// TwinCAT 3 PLC project DemoPLC
// ProgramVersion: 3.1.4020.1
// libraries:
//   Tc2_Drive, * (Beckhoff Automation GmbH)
//   Tc2_EtherCAT, * (Beckhoff Automation GmbH)
//   Tc2_Math, * (Beckhoff Automation GmbH)
//   Tc2_MC2, * (Beckhoff Automation GmbH)
//   Tc2_MC2_Drive, * (Beckhoff Automation GmbH)
//   Tc2_MDP, * (Beckhoff Automation GmbH)
//   Tc2_Smtp, * (Beckhoff Automation GmbH)
//   Tc2_Standard, * (Beckhoff Automation GmbH)
//   Tc2_System, * (Beckhoff Automation GmbH)
//   Tc2_Utilities, * (Beckhoff Automation GmbH)
//   Tc3_Module, * (Beckhoff Automation GmbH)
// project tree:
//   DUTs/DataAndTime/ E_DayPL.TcDUT, E_DayPLShort.TcDUT, E_Location.TcDUT, E_MonthPL.TcDUT, E_SeasonPL.TcDUT, ST_Calendar.TcDUT, ST_ConstHoliday.TcDUT, ST_ConstLocation.TcDUT, ST_Holiday.TcDUT, ST_Location.TcDUT
//   DUTs/ GEN_MODE.TcDUT, NEWTYPE.TcDUT, ST_AX5000_Diag_MC2.TcDUT, ST_EL3403_Data.TcDUT, ST_KL3403_Report.TcDUT, ST_STRING_2040.TcDUT
//   / MAIN.TcPOU, PlcTask.TcTTO
//   POUs/Blinkers/ FB_Blink_AS.TcPOU, FB_Blink_S.TcPOU
//   POUs/Conversions/ ArrayOfReal_To_String.TcPOU, arrBOOL16_TO_WORD.TcPOU, arrBOOL8_TO_BYTE.TcPOU, ArrOfInt_To_String.TcPOU, FB_CONCAT_S2040.TcPOU, FB_IntTo2Byte.TcPOU, F_4BYTES_TO_DWORD.TcPOU, F_4BYTES_TO_REAL.TcPOU, F_8BYTES_TO_LREAL.TcPOU, F_BCDToDec.TcPOU, F_CLEAN_S2040.TcPOU, F_Convert_4BBCD_To_Real.TcPOU, F_DWORD_TO_REAL.TcPOU, F_Words_to_Real.TcPOU, GRAYB_TO_WORD.TcPOU, GRAYW_TO_WORD.TcPOU
//   POUs/Conversions/BitOriented/ BCD_TO_INT.TcPOU, F_1stByteW.TcPOU, F_1stByteWtoB.TcPOU, F_2Bytes_To_Word.TcPOU, F_2ndByteW.TcPOU, F_2ndByteWtoB.TcPOU, F_MaskWord.TcPOU, L_TBConvArrBitsToDword.TcPOU, L_TBConvBitsToByte.TcPOU, L_TBConvBitsToDword.TcPOU, L_TBConvBitsToWord.TcPOU, L_TBConvByteToBits.TcPOU, L_TBConvDwordToArrBits.TcPOU, L_TBConvDwordToBits.TcPOU, L_TBConvWordToBits.TcPOU, L_TBGetBitOfByte.TcPOU, L_TBGetBitOfDword.TcPOU, L_TBGetBitOfWord.TcPOU, L_TBResetBitOfByte.TcPOU, L_TBResetBitOfDword.TcPOU, L_TBResetBitOfWord.TcPOU, L_TBSetBitOfByte.TcPOU, L_TBSetBitOfDword.TcPOU, L_TBSetBitOfWord.TcPOU, L_TBSquareWave.TcPOU
//   POUs/DateAndTime/ FB_AstrTimeCET.TcPOU, FB_CycleTime.TcPOU, FB_DST.TcPOU, FB_GetSystemTime.TcPOU, FB_Period.TcPOU, FB_PolishPublicHoliday.TcPOU, FB_SimpleWorkTime.TcPOU, FB_TimeMeasure.TcPOU, FB_TimeMeasureEx.TcPOU, FB_WeekSchedule.TcPOU, FB_Worktime.TcPOU, FB_WorktimeCompact.TcPOU, F_DT_To_sDT_Ind.TcPOU, F_ExcelDateMin.TcPOU, F_ExcelDateSec.TcPOU, F_sDT_Ind_To_DT.TcPOU
//   POUs/EL_Terminals/ FB_EL3403.TcPOU, FB_EL3403Ex.TcPOU, FB_EL3403Ex2.TcPOU
//   POUs/FileAccess/ FB_EmailLog.TcPOU, FB_FileLog.TcPOU, FB_FilePutText.TcPOU, FB_ReceipRW.TcPOU, FB_SaveLineToFile.TcPOU, FB_SaveTextToFile.TcPOU (not stored), FB_WriteReportToFile.TcPOU, FB_XCopyCE.TcPOU
//   POUs/FlipFlop/ FB_toggle.TcPOU, FB_TOGGLE_WITH_RESET.TcPOU, FB_TypeJK.TcPOU, FB_TypeJK_SEL.TcPOU, FB_TypeRS.TcPOU, FB_TypeSR.TcPOU
//   POUs/HVAC/ FB_AirMixer.TcPOU, FB_Alarm.TcPOU, FB_Boiler_Load.TcPOU, FB_Controller2Point.TcPOU, FB_DeadNullRange.TcPOU, FB_LimitHVAC.TcPOU, FB_SeqCMH.TcPOU
//   POUs/KL_Terminals/ FB_KL320x_1channel.TcPOU, FB_KL32x8_1channel.TcPOU, FB_KL32x8_1channelEx.TcPOU, FB_KL3403_1channel.TcPOU, FB_PowerMeasuring.TcPOU
//   POUs/NC/ FB_AX5000_Diag_MC2.TcPOU, FB_AxisParameter.TcPOU, FB_CalculateSpeed.TcPOU, FB_Enc20bitToDWORD.TcPOU, FB_EncIntToDint.TcPOU, FB_EncWordtoDword.TcPOU, FB_ForceLockUnlock.TcPOU, FB_I2T_AX2000.TcPOU, FB_I2T_EL72x1.TcPOU, FB_PWM_BASIC.TcPOU, FB_SetBiasValue.TcPOU, FB_TorqueMonitoringEL_Ex2.TcPOU, FB_TorqueMonitoringEx2.TcPOU
//   POUs/Switches/ FB_2SwB.TcPOU, FB_2SwM.TcPOU, FB_Click.TcPOU, FB_ClickCounterBit.TcPOU, FB_ClickCounterByte.TcPOU, FB_Dimmer1P.TcPOU, FB_Dimmer1PMinMax.TcPOU, FB_Dimmer2P.TcPOU, FB_Dimmer2PMinMax.TcPOU, FB_ShortLong.TcPOU, FB_ShortLongTrig.TcPOU, FB_Sw4F.TcPOU, FB_Sw4FTrig.TcPOU, FB_SwOrSen.TcPOU, FB_SwOrSenTrig.TcPOU
//   POUs/Various/ FB_AnalogTo3Point.TcPOU, FB_Average.TcPOU, FB_CERHOST.TcPOU, FB_DiskFreeSpace.TcPOU, FB_Filter.TcPOU, FB_FilterEx.TcPOU, FB_Generator.TcPOU, FB_Hysteresis.TcPOU, FB_Persistent.TcPOU, FB_PIDBasic.TcPOU, FB_Ramp.TcPOU, FB_ReadRegister.TcPOU, FB_RecMove.TcPOU, FB_SetIPAddress.TcPOU, FB_SinGenerator.TcPOU, FB_WriteRegister.TcPOU, F_CRC_CALC.TcPOU, F_ScaleLREAL.TcPOU, F_Scaling.TcPOU (not stored), TIMER.TcPOU, TONR.TcPOU
// real-time tasks:
//   TASK PlcTask: cycle T#10ms, priority 20, ADS port 350

CONFIGURATION DemoPLC
    RESOURCE PLC ON TwinCAT3
        TASK PlcTask(INTERVAL := T#10ms, PRIORITY := 20);
        PROGRAM MAIN WITH PlcTask : MAIN;
    END_RESOURCE
END_CONFIGURATION

// ---- DUTs/DataAndTime/E_DayPL.TcDUT
TYPE E_DayPL :(Poniedzialek:=1, Wtorek, Sroda, Czwartek, Piatek, Sobota, Niedziela );
END_TYPE

// ---- DUTs/DataAndTime/E_DayPLShort.TcDUT
TYPE E_DayPLShort :(Pn:=1, Wt, SR, Cz, Pt, So, N);
END_TYPE

// ---- DUTs/DataAndTime/E_Location.TcDUT
TYPE E_Location : (Wroclaw:=1, Warszawa, Krakow, Zakopane, Katowice, Poznan );
END_TYPE

// ---- DUTs/DataAndTime/E_MonthPL.TcDUT
TYPE E_MonthPL :(Stycznen:=1, Luty, Marzec, Kwiecien, Maj,  Czerwiec, Lipiec, Sierpien, Wrzesien, Pazdziernik, Listopad, Grudzien);
END_TYPE

// ---- DUTs/DataAndTime/E_SeasonPL.TcDUT
TYPE E_SeasonPL : (Wiosna:=1, Lato, Jesien, Zima);
END_TYPE

// ---- DUTs/DataAndTime/ST_Calendar.TcDUT
TYPE ST_Calendar :
STRUCT
	dateDate : DATE;				(* data *)
	wYear : WORD;				(* rok  *)
	wMonth : WORD;				(* miesiąc  *)
	wDay : WORD;				(* dzień *)
	bLeapYear: BOOL;			(* true if rok przestępny *)
	eWeekDay: E_DayPL;			(* dzień tygodnia *)
	wNoWeek : WORD;			(* nr tygodnia w roku *)
	wDayInYear: WORD;			(* nr dnia w roku *)
	bHoliday : BOOL;				(* true jesli jest swieto *)
	sHolidayName: STRING(30);	(* nazwa swieta *)
	eSeason: E_SeasonPL;		(* pora roku *)
	sLocation: STRING(30);		(* lokalizacja *)
	rLatitude: REAL;				(* szerokosc geograficzna np. Wrocław :=51.1174 *) (* do obliczen wschodu i zachodu slonca *)
	rLongitude: REAL;				(* długosc geograficzna np. Wrocław := 17.0383 *)
	todSunRise: TOD;				(* sun_rise for current location *)
	todSunSet : TOD;				(* sun_set for current location *)
END_STRUCT
END_TYPE

// ---- DUTs/DataAndTime/ST_ConstHoliday.TcDUT
TYPE ST_ConstHoliday :
STRUCT
	// Zapamietane dni swiat 
	//  gc_ConstHoliday - rozmiar tablicy array of ST_Holiday size   -> Var_Global_Calendar;   
	//  w tablicy najpierw nalezy podac swieta stale 
	//  if month = 0 obliczamy swieto ruchome
	//  iExecute mowi ile dni wczesniej/pozniej jest swieto
	astLocation: ARRAY [1..15] OF ST_Holiday := [		(sName := 'Nowy Rok', 				wDay := 1, 	wMonth := 1),
														(sName := 'Swieto Pracy', 			wDay := 1, 	wMonth := 5),
														(sName := 'Konstytucja 3 Maja', 	wDay := 3, 	wMonth := 5),
														(sName := 'Wniebowstapienie NMP',	wDay := 15,	wMonth := 8),
														(sName := 'Wszystkich Swietych', 	wDay := 1, 	wMonth := 11),
														(sName := 'Swieto Niepodleglosc', 	wDay := 11, 	wMonth := 11),
														(sName := 'Boze Narodzenie', 		wDay := 25, 	wMonth := 12),
														(sName := 'Boze Narodzenie', 		wDay := 26, 	wMonth := 12),
														(sName := 'Wielki Piatek',			wDay := 0, 	wMonth := 0, iExecute := -2),
														(sName := 'Wielka Sobota', 			wDay := 0, 	wMonth := 0, iExecute := -1),
														(sName := 'Wielkanoc', 				wDay := 0, 	wMonth := 0, iExecute := 0),
														(sName := 'Poniedziałek Wielkanocny', wDay :=1,	wMonth := 0, iExecute := 1),
														(sName := 'Boze Cialo', 			wDay := 0, 	wMonth := 0, iExecute := 60),
														2(())];
END_STRUCT
END_TYPE

// ---- DUTs/DataAndTime/ST_ConstLocation.TcDUT
TYPE ST_ConstLocation :
STRUCT
	(* to memorize location *)
	(* gc_ConstLocation - max array of ST_Location  size  -> Var_Global_Calendar;   *)
	astLocation : ARRAY [1.. 10] OF ST_Location := [(sName := 'Wroclaw', rLatitude := 51.1174, rLongitude := 17.0383),
											(sName := 'Warszawa', rLatitude := 52.248, rLongitude := 21.008),
											(sName := 'Krakow', rLatitude := 50.085, rLongitude := 19.940),
											(sName := 'Zakopane', rLatitude := 49.3091, rLongitude := 19.9524),
											(sName := 'Katowice', rLatitude := 50.2746, rLongitude := 19.0255),
											(sName := 'Poznan', rLatitude := 52.425, rLongitude :=  16.927),
											(),
											(),
											(),
											()];

END_STRUCT
END_TYPE

// ---- DUTs/DataAndTime/ST_Holiday.TcDUT
TYPE ST_Holiday :
STRUCT
	sName : STRING(30); 	(* holiday's name *)
	wDay : WORD ;		(* holiday's day, part of date *)
	wMonth : WORD;		(* holiday's month, part of date *)
	iExecute : INT;		(* 0 - nie swietujemy, -1 = dzien wczesniej, +1 = dzien pozniej *)
END_STRUCT
END_TYPE

// ---- DUTs/DataAndTime/ST_Location.TcDUT
TYPE ST_Location :
STRUCT
	sName: STRING(30); 	(* location's name ex. Wroclaw*)
	rLatitude: REAL;		(* szerokosc geograficzna np. Wrocław :=51.1174 *)
	rLongitude: REAL;		(* długosc geograficzna np. Wrocław := 17.0383 *)
END_STRUCT
END_TYPE

// ---- DUTs/GEN_MODE.TcDUT
TYPE GEN_MODE :
	(TRIANGLE:=0,TRIANGLE_POS:=1,SAWTOOTH_RISE:=2,SAWTOOTH_FALL:=3,RECTANGLE:=4,SINUS:=5,COSINUS:=6);
END_TYPE

// ---- DUTs/NEWTYPE.TcDUT
TYPE NEWTYPE :
STRUCT
	No1: STRING;
	No2: INT;
	No3: BOOL;
END_STRUCT
END_TYPE

// ---- DUTs/ST_AX5000_Diag_MC2.TcDUT
TYPE ST_AX5000_Diag_MC2 :
STRUCT
	nClass1_Diagnostic : WORD;
	nDiagNumber: UDINT;
	nDC_Bus_Voltage: REAL;
	nDC_Bus_Current: REAL;
	nDrive_Temp: REAL;
	nMotor_Temp: REAL;
	sDiagnosticMessage: STRING;
	DiagList: ST_SoE_DiagNumList;
END_STRUCT
END_TYPE

// ---- DUTs/ST_EL3403_Data.TcDUT
TYPE ST_EL3403_Data :
STRUCT
	rCurrent1				: REAL; (* Unit 1 A *)
	rCurrent2				: REAL; (* Unit 1 A *)
	rCurrent3				: REAL; (* Unit 1 A *)
	rVoltage1				: REAL; (* Unit 1 V *)
	rVoltage2				: REAL; (* Unit 1 V *)
	rVoltage3				: REAL; (* Unit 1 V *)
	rActivePower1			: REAL; (* Unit 1 W *)
	rActivePower2			: REAL; (* Unit 1 W *)
	rActivePower3			: REAL; (* Unit 1 W *)
	rApparentPower1		: REAL; (* Unit 1 VA *)
	rApparentPower2		: REAL; (* Unit 1 VA *)
	rApparentPower3		: REAL; (* Unit 1 VA *)
	rReactivePower1		: REAL; (* Unit 1 VAR *)
	rReactivePower2		: REAL; (* Unit 1 VAR *)
	rReactivePower3		: REAL; (* Unit 1 VAR *)
	rEnergy1				: REAL; (* Unit 1 Wh *)
	rEnergy2				: REAL; (* Unit 1 Wh *)
	rEnergy3				: REAL; (* Unit 1 Wh *)
	rCosPhi1				: REAL; (* Unit 1 *)
	rCosPhi2				: REAL; (* Unit 1 *)
	rCosPhi3				: REAL; (* Unit 1 *)
	rFrequency1			: REAL; (* Unit 1 Hz *)
	rFrequency2			: REAL; (* Unit 1 Hz *)
	rFrequency3			: REAL; (* Unit 1 Hz *)
	rEnergyNegative1		: REAL; (* Unit 1 Wh *)
	rEnergyNegative2		: REAL; (* Unit 1 Wh *)
	rEnergyNegative3		: REAL; (* Unit 1 Wh *)
END_STRUCT
END_TYPE

// ---- DUTs/ST_KL3403_Report.TcDUT
TYPE ST_KL3403_Report :
STRUCT
	Summary: WORD;
	SummaryPrice:WORD;
	Tarrif1: WORD;
	Tarrif1Price:WORD;
	Tarrif2: WORD;
	Tarrif2Price:WORD;
END_STRUCT
END_TYPE

// ---- DUTs/ST_STRING_2040.TcDUT
TYPE
	ST_STRING_2040 :  ARRAY[1..8] OF STRING(255);
END_TYPE

// ---- MAIN.TcPOU
//==================================================================================================
//					Beckhoff Automation Poland
//							30.05.2017
//	v1.3	|| TC v 3.1.4020.32		|| dodany blok NC\FB_AxisParameter
//	v1.2	|| TC v 3.1.4020.32		|| dodany blok Various\FB_AnalogTo3Point
//	v1.1	|| TC v 3.1.4020.28		|| dodany blok Various\FB_PIDBasic
//									|| dodany blok Various\FB_SinGenerator
// 	v1.0 	|| TC v 3.1.4020.28 	|| pierwsza wersja
//==================================================================================================
PROGRAM MAIN
VAR
END_VAR

END_PROGRAM

// ---- POUs/Blinkers/FB_Blink_AS.TcPOU
(********************************************************************************************)
(*							Beckhoff Automation Poland										*)
(*								FB_Blink_AS	 v1.1											*)
(*									9.11.2007												*)
(*						Blok funkcyjny zegara asynchronicznego								*)
(*__________________________________________________________________________________________*)

FUNCTION_BLOCK FB_Blink_AS
VAR_INPUT
	T1										:	TIME;				(*Czas, gdy wyjście przyjmuje wartość TRUE*)
	T0										:	TIME;				(*Czas, gdy wyjście przyjmuje wartość FALSE*)
END_VAR
VAR_OUTPUT
	Q										:	BOOL;				(*Wyjscie*)
END_VAR
VAR
	ton1									:	TON;
	ton2									:	TON;
END_VAR

ton1(IN:= NOT ton2.Q, PT:=T0);
Q:=ton1.Q;
ton2(IN:=ton1.Q , PT:=T1);

END_FUNCTION_BLOCK

// ---- POUs/Blinkers/FB_Blink_S.TcPOU
(********************************************************************************************)
(*							Beckhoff Automation Poland										*)
(*								FB_Blink_S	 v1.1											*)
(*									9.11.2007												*)
(*						Blok funkcyjny zegara synchronicznego								*)
(*__________________________________________________________________________________________*)

FUNCTION_BLOCK FB_Blink_S
VAR_INPUT
	Tv										:	TIME;				(*Czas trwania impulsu i przerwy*)
END_VAR
VAR_OUTPUT
	Q										:	BOOL;				(*Wyjscie*)
END_VAR
VAR
	ton1									:	TON;
	ton2									:	TON;
END_VAR

ton1(IN:= NOT ton2.Q, PT:=Tv);
Q:=ton1.Q;
ton2(IN:=ton1.Q , PT:=ton1.PT );

END_FUNCTION_BLOCK

// ---- POUs/Conversions/ArrayOfReal_To_String.TcPOU
(****************************************************************************************)
(*							Beckhoff Automation Poland									*)
(*							ArrayOfReal_To_String	 v1.2								*)
(*									30.12.2009											*)
(*								v1.2 - dynamiczny rozmiar tablic						*)
(*		Funkcja konwerująca tablicę zmiennych typu REAL na zmienną typu STRING(255)		*)
(*		Zmienne typu REAL oddzielone są znakiem tabulacji ($t)							*)
(*		Powstały napis nie posiada znaku końca linii ($n)								*)
(*		Uwaga!!																			*)
(*		Należy zwrócić uwagę na ilość znaków przypadającą na każdą zmienną typu REAL	*)
(*______________________________________________________________________________________*)

FUNCTION ArrayOfReal_To_String: STRING(255)
VAR_INPUT
	pData: POINTER TO REAL;
	Length : 	UDINT;
END_VAR
VAR
	pos : UDINT;
	bBusy: BOOL;
	sTemp: STRING(7);
	rTemp: REAL;
END_VAR

pos := 1;
REPEAT
	IF pos > Length THEN
		bBusy := FALSE;
	ELSE
		rTemp := pData^;
		sTemp := LREAL_TO_FMTSTR(rTemp,2,TRUE);
		ArrayOfReal_To_String := CONCAT( ArrayOfReal_To_String,CONCAT(sTemp,'$t'));
		pos := pos + 4;
		(* increment pointer *)
		pData := pData+4;
		bBusy := TRUE;
	END_IF
UNTIL  NOT bBusy
END_REPEAT

END_FUNCTION

// ---- POUs/Conversions/arrBOOL16_TO_WORD.TcPOU
(************************************************************************************)
(*							Beckhoff Automation Poland								*)
(*								arrBOOL16_TO_WORD v1.0								*)
(*									15.02.2010										*)
(*		Funkcja tworząca zmienną typu WORD z tablicy 16 zmiennych typu BOOL			*)
(*__________________________________________________________________________________*)
FUNCTION arrBOOL16_TO_WORD : WORD
VAR_INPUT
	aBool16 : ARRAY [0..15] OF BOOL;
END_VAR

arrBOOL16_TO_WORD.0 := aBool16[0];
arrBOOL16_TO_WORD.1 := aBool16[1];
arrBOOL16_TO_WORD.2 := aBool16[2];
arrBOOL16_TO_WORD.3 := aBool16[3];
arrBOOL16_TO_WORD.4 := aBool16[4];
arrBOOL16_TO_WORD.5 := aBool16[5];
arrBOOL16_TO_WORD.6 := aBool16[6];
arrBOOL16_TO_WORD.7 := aBool16[7];
arrBOOL16_TO_WORD.8 := aBool16[8];
arrBOOL16_TO_WORD.9 := aBool16[9];
arrBOOL16_TO_WORD.10 := aBool16[10];
arrBOOL16_TO_WORD.11 := aBool16[11];
arrBOOL16_TO_WORD.12 := aBool16[12];
arrBOOL16_TO_WORD.13 := aBool16[13];
arrBOOL16_TO_WORD.14 := aBool16[14];
arrBOOL16_TO_WORD.15 := aBool16[15];

END_FUNCTION

// ---- POUs/Conversions/arrBOOL8_TO_BYTE.TcPOU
(****************************************************************************************)
(*							Beckhoff Automation Poland									*)
(*								arrBOOL8_TO_BYTE v1.0									*)
(*									15.02.2010											*)
(*		Funkcja tworząca zmienną typu BYTE z tablicy 8 zmiennych typu BOOL				*)
(*______________________________________________________________________________________*)
FUNCTION arrBOOL8_TO_BYTE : BYTE
VAR_INPUT
	aBool8 : ARRAY [0..7] OF BOOL;
END_VAR

arrBOOL8_TO_BYTE.0 := aBool8[0];
arrBOOL8_TO_BYTE.1 := aBool8[1];
arrBOOL8_TO_BYTE.2 := aBool8[2];
arrBOOL8_TO_BYTE.3 := aBool8[3];
arrBOOL8_TO_BYTE.4 := aBool8[4];
arrBOOL8_TO_BYTE.5 := aBool8[5];
arrBOOL8_TO_BYTE.6 := aBool8[6];
arrBOOL8_TO_BYTE.7 := aBool8[7];

END_FUNCTION

// ---- POUs/Conversions/ArrOfInt_To_String.TcPOU
(****************************************************************************************)
(*							Beckhoff Automation Poland									*)
(*								ArrOfInt_To_String	 v1.2								*)
(*								30.12.2009												*)
(*								v1.2 - dynamiczny rozmiar tablic						*)
(*		Funkcja konwerująca tablicę zmiennych typu INT na zmienną typu STRING(255)		*)
(*		Zmienne typu INT oddzielone są znakiem tabulacji ($t)							*)
(*		Powstały napis nie posiada znaku końca linii ($n)								*)
(*______________________________________________________________________________________*)

FUNCTION ArrOfInt_To_String : STRING(255)
VAR_INPUT
	pData: POINTER TO INT;
	Length : 	UDINT;
END_VAR
VAR
	pos : UDINT;
	bBusy: BOOL;
	iTemp: INT;
END_VAR

pos := 1;
REPEAT
	IF pos > Length THEN
		bBusy := FALSE;
	ELSE
		iTemp := pData^;
		ArrOfInt_To_String := CONCAT(ArrOfInt_To_String,CONCAT(INT_TO_STRING(iTemp),'$t'));
		pos := pos + 2;
		(* increment pointer *)
		pData := pData+2;
		bBusy := TRUE;
	END_IF
UNTIL  NOT bBusy
END_REPEAT

END_FUNCTION

// ---- POUs/Conversions/BitOriented/BCD_TO_INT.TcPOU
(********************************************************************************************)
(*							Beckhoff Automation Poland										*)
(*								FB_BCD_TO_INT	 v1.0										*)
(*									26.06.2008												*)
(*		Funkcja zamieniająca liczbę w formacie BCD na wartość typu integer. 	   			*)
(*		Gdy na wejście funkcji zostanie wprowadzona zła wartość funkcja zwróci wartość  -1	*)
(*__________________________________________________________________________________________*)


FUNCTION BCD_TO_INT : INT	(* Funkcja zwraca wartość typu INT*)
VAR_INPUT
	B:BYTE;					(* Zmienna wejściowa typu Byte*)
END_VAR

IF SHR(B,4)>9 OR B-SHL(SHR(B,4),4)>9 THEN
	BCD_TO_INT:=-1;
ELSE
	BCD_TO_INT:=B-SHR(B,4)*6;
END_IF;

END_FUNCTION

// ---- POUs/Conversions/BitOriented/F_1stByteW.TcPOU
(****************************************************************************************)
(*							Beckhoff Automation Poland									*)
(*									F_1stByteW	v1.0									*)
(*									15.02.2010											*)
(*		Funkcja wyciagajaca mniej znaczacy BYTE ze zmiennej typu WORD					*)
(*							 wyjscie typu WORD											*)
(*______________________________________________________________________________________*)
FUNCTION F_1stByteW : WORD
VAR_INPUT
	wIn:	WORD;
END_VAR

F_1stByteW := wIn AND 16#FF;

END_FUNCTION

// ---- POUs/Conversions/BitOriented/F_1stByteWtoB.TcPOU
(****************************************************************************************)
(*							Beckhoff Automation Poland									*)
(*								F_1stByteWtoB v1.0										*)
(*									15.02.2010											*)
(*		Funkcja wyciagajaca mniej znaczacy BYTE ze zmiennej typu WORD					*)
(*							 wyjscie typu BYTE											*)
(*______________________________________________________________________________________*)
FUNCTION F_1stByteWtoB : BYTE
VAR_INPUT
	wIn		:	WORD;
END_VAR

F_1stByteWtoB := WORD_TO_BYTE(wIn AND 16#FF);

END_FUNCTION

// ---- POUs/Conversions/BitOriented/F_2Bytes_To_Word.TcPOU
(****************************************************************************************)
(*							Beckhoff Automation Poland									*)
(*								F_2Bytes_To_Word v1.0									*)
(*									15.02.2010											*)
(*		Funkcja tworząca zmienną typu WORD z dwóch zmiennych typu BYTE					*)
(*______________________________________________________________________________________*)
FUNCTION F_2Bytes_To_Word : WORD
VAR_INPUT
	byHigh	:	BYTE;
	byLow	:	BYTE;
END_VAR
VAR
END_VAR

F_2Bytes_To_Word := byHigh;
F_2Bytes_To_Word := SHL(F_2Bytes_To_Word,8);
F_2Bytes_To_Word := F_2Bytes_To_Word + byLow;

END_FUNCTION

// ---- POUs/Conversions/BitOriented/F_2ndByteW.TcPOU
(****************************************************************************************)
(*							Beckhoff Automation Poland									*)
(*								F_2ndByteW v1.0											*)
(*									15.02.2010											*)
(*		Funkcja wyciagajaca bardziej znaczacy BYTE ze zmiennej typu WORD				*)
(*							 wyjscie typu WORD											*)
(*______________________________________________________________________________________*)
FUNCTION F_2ndByteW : WORD
VAR_INPUT
	wIn		:	WORD;
END_VAR

F_2ndByteW := wIn AND 16#FF00;

END_FUNCTION

// ---- POUs/Conversions/BitOriented/F_2ndByteWtoB.TcPOU
(****************************************************************************************)
(*							Beckhoff Automation Poland									*)
(*								F_2ndByteWtoB v1.0										*)
(*									15.02.2010											*)
(*		Funkcja wyciagajaca bardziej znaczacy BYTE ze zmiennej typu WORD				*)
(*							 	wyjscie typu BYTE										*)
(*______________________________________________________________________________________*)
FUNCTION F_2ndByteWtoB : BYTE
VAR_INPUT
	wIn		:	WORD;
END_VAR

F_2ndByteWtoB := WORD_TO_BYTE(SHR(wIn,8));

END_FUNCTION

// ---- POUs/Conversions/BitOriented/F_MaskWord.TcPOU
(****************************************************************************************)
(*							Beckhoff Automation Poland									*)
(*								F_MaskWord v1.0											*)
(*									15.02.2010											*)
(*		Funkcja wyciagajaca  okreslona ilosc Bitow ze ze zmiennej typu WORD				*)
(*							 wyjscie typu WORD											*)
(*______________________________________________________________________________________*)
FUNCTION F_MaskWord : WORD
VAR_INPUT
	wIn	:	WORD; (*Wejscie*)
	wNo	:	WORD; (*Ilosc bitow, zaczynajac od LSB*)
END_VAR

CASE wNo OF
	0:
	F_MaskWord := wIn AND 2#0;
	1:
	F_MaskWord := wIn AND 2#1;
	2:
	F_MaskWord := wIn AND 2#11;
	3:
	F_MaskWord := wIn AND 2#111;
	4:
	F_MaskWord := wIn AND 2#1111;
	5:
	F_MaskWord := wIn AND 2#11111;
	6:
	F_MaskWord := wIn AND 2#111111;
	7:
	F_MaskWord := wIn AND 2#1111111;
	8:
	F_MaskWord := wIn AND 2#11111111;
	9:
	F_MaskWord := wIn AND 2#111111111;
	10:
	F_MaskWord := wIn AND 2#1111111111;
	11:
	F_MaskWord := wIn AND 2#11111111111;
	12:
	F_MaskWord := wIn AND 2#111111111111;
	13:
	F_MaskWord := wIn AND 2#1111111111111;
	14:
	F_MaskWord := wIn AND 2#11111111111111;
	15:
	F_MaskWord := wIn AND 2#111111111111111;
	16:
	F_MaskWord := wIn;
END_CASE

END_FUNCTION

// ---- POUs/Conversions/BitOriented/L_TBConvArrBitsToDword.TcPOU
(****************************************************************************************)
(*							Beckhoff Automation Poland									*)
(*							L_TBConvArrBitsToDword  v1.0								*)
(*									7.04.2009											*)
(*		This function converts array 32 single bits into a value of type ”double word”	*)
(*______________________________________________________________________________________*)
FUNCTION L_TBConvArrBitsToDword : DWORD
VAR_INPUT
	arrBits: ARRAY [0..31] OF BOOL;
END_VAR

L_TBConvArrBitsToDword.0 := arrBits[0];
L_TBConvArrBitsToDword.1 := arrBits[1];
L_TBConvArrBitsToDword.2 := arrBits[2];
L_TBConvArrBitsToDword.3 := arrBits[3];
L_TBConvArrBitsToDword.4 := arrBits[4];
L_TBConvArrBitsToDword.5 := arrBits[5];
L_TBConvArrBitsToDword.6 := arrBits[6];
L_TBConvArrBitsToDword.7 := arrBits[7];
L_TBConvArrBitsToDword.8 := arrBits[8];
L_TBConvArrBitsToDword.9 := arrBits[9];
L_TBConvArrBitsToDword.10 := arrBits[10];
L_TBConvArrBitsToDword.11 := arrBits[11];
L_TBConvArrBitsToDword.12 := arrBits[12];
L_TBConvArrBitsToDword.13 := arrBits[13];
L_TBConvArrBitsToDword.14 := arrBits[14];
L_TBConvArrBitsToDword.15 := arrBits[15];
L_TBConvArrBitsToDword.16 := arrBits[16];
L_TBConvArrBitsToDword.17 := arrBits[17];
L_TBConvArrBitsToDword.18 := arrBits[18];
L_TBConvArrBitsToDword.19 := arrBits[19];
L_TBConvArrBitsToDword.20 := arrBits[20];
L_TBConvArrBitsToDword.21 := arrBits[21];
L_TBConvArrBitsToDword.22 := arrBits[22];
L_TBConvArrBitsToDword.23 := arrBits[23];
L_TBConvArrBitsToDword.24 := arrBits[24];
L_TBConvArrBitsToDword.25 := arrBits[25];
L_TBConvArrBitsToDword.26 := arrBits[26];
L_TBConvArrBitsToDword.27 := arrBits[27];
L_TBConvArrBitsToDword.28 := arrBits[28];
L_TBConvArrBitsToDword.29 := arrBits[29];
L_TBConvArrBitsToDword.30 := arrBits[30];
L_TBConvArrBitsToDword.31 := arrBits[31];

END_FUNCTION

// ---- POUs/Conversions/BitOriented/L_TBConvBitsToByte.TcPOU
(****************************************************************************************)
(*							Beckhoff Automation Poland									*)
(*							L_TBConvBitsToByte 	 v1.0									*)
(*									29.02.2007											*)
(*			This function converts 8 single bit values into a value of type ”byte”		*)
(*______________________________________________________________________________________*)
FUNCTION L_TBConvBitsToByte : BYTE
VAR_INPUT
	bBit0: BOOL;
	bBit1: BOOL;
	bBit2: BOOL;
	bBit3: BOOL;
	bBit4: BOOL;
	bBit5: BOOL;
	bBit6: BOOL;
	bBit7: BOOL;
END_VAR

L_TBConvBitsToByte.0 := bBit0;
L_TBConvBitsToByte.1 := bBit1;
L_TBConvBitsToByte.2 := bBit2;
L_TBConvBitsToByte.3 := bBit3;
L_TBConvBitsToByte.4 := bBit4;
L_TBConvBitsToByte.5 := bBit5;
L_TBConvBitsToByte.6 := bBit6;
L_TBConvBitsToByte.7 := bBit7;

END_FUNCTION

// ---- POUs/Conversions/BitOriented/L_TBConvBitsToDword.TcPOU
(****************************************************************************************)
(*							Beckhoff Automation Poland									*)
(*							L_TBConvBitsToDword  v1.0									*)
(*									29.02.2007											*)
(*		This function converts 32 single bit values into a value of type ”double word”	*)
(*______________________________________________________________________________________*)
FUNCTION L_TBConvBitsToDword : DWORD
VAR_INPUT
	bBit0: BOOL;
	bBit1: BOOL;
	bBit2: BOOL;
	bBit3: BOOL;
	bBit4: BOOL;
	bBit5: BOOL;
	bBit6: BOOL;
	bBit7: BOOL;
	bBit8: BOOL;
	bBit9: BOOL;
	bBit10: BOOL;
	bBit11: BOOL;
	bBit12: BOOL;
	bBit13: BOOL;
	bBit14: BOOL;
	bBit15: BOOL;
	bBit16: BOOL;
	bBit17: BOOL;
	bBit18: BOOL;
	bBit19: BOOL;
	bBit20: BOOL;
	bBit21: BOOL;
	bBit22: BOOL;
	bBit23: BOOL;
	bBit24: BOOL;
	bBit25: BOOL;
	bBit26: BOOL;
	bBit27: BOOL;
	bBit28: BOOL;
	bBit29: BOOL;
	bBit30: BOOL;
	bBit31: BOOL;
END_VAR

L_TBConvBitsToDword.0 := bBit0;
L_TBConvBitsToDword.1 := bBit1;
L_TBConvBitsToDword.2 := bBit2;
L_TBConvBitsToDword.3 := bBit3;
L_TBConvBitsToDword.4 := bBit4;
L_TBConvBitsToDword.5 := bBit5;
L_TBConvBitsToDword.6 := bBit6;
L_TBConvBitsToDword.7 := bBit7;
L_TBConvBitsToDword.8 := bBit8;
L_TBConvBitsToDword.9 := bBit9;
L_TBConvBitsToDword.10 := bBit10;
L_TBConvBitsToDword.11 := bBit11;
L_TBConvBitsToDword.12 := bBit12;
L_TBConvBitsToDword.13 := bBit13;
L_TBConvBitsToDword.14 := bBit14;
L_TBConvBitsToDword.15 := bBit15;
L_TBConvBitsToDword.16 := bBit16;
L_TBConvBitsToDword.17 := bBit17;
L_TBConvBitsToDword.18 := bBit18;
L_TBConvBitsToDword.19 := bBit19;
L_TBConvBitsToDword.20 := bBit20;
L_TBConvBitsToDword.21 := bBit21;
L_TBConvBitsToDword.22 := bBit22;
L_TBConvBitsToDword.23 := bBit23;
L_TBConvBitsToDword.24 := bBit24;
L_TBConvBitsToDword.25 := bBit25;
L_TBConvBitsToDword.26 := bBit26;
L_TBConvBitsToDword.27 := bBit27;
L_TBConvBitsToDword.28 := bBit28;
L_TBConvBitsToDword.29 := bBit29;
L_TBConvBitsToDword.30 := bBit30;
L_TBConvBitsToDword.31 := bBit31;

END_FUNCTION

// ---- POUs/Conversions/BitOriented/L_TBConvBitsToWord.TcPOU
(****************************************************************************************)
(*							Beckhoff Automation Poland									*)
(*							L_TBConvBitsToWord  v1.0									*)
(*									29.02.2007											*)
(*			This function converts 16 single bit values into a value of type ”word”		*)
(*______________________________________________________________________________________*)
FUNCTION L_TBConvBitsToWord : WORD
VAR_INPUT
	bBit0: BOOL;
	bBit1: BOOL;
	bBit2: BOOL;
	bBit3: BOOL;
	bBit4: BOOL;
	bBit5: BOOL;
	bBit6: BOOL;
	bBit7: BOOL;
	bBit8: BOOL;
	bBit9: BOOL;
	bBit10: BOOL;
	bBit11: BOOL;
	bBit12: BOOL;
	bBit13: BOOL;
	bBit14: BOOL;
	bBit15: BOOL;
END_VAR
VAR
END_VAR

L_TBConvBitsToWord.0 := bBit0;
L_TBConvBitsToWord.1 := bBit1;
L_TBConvBitsToWord.2 := bBit2;
L_TBConvBitsToWord.3 := bBit3;
L_TBConvBitsToWord.4 := bBit4;
L_TBConvBitsToWord.5 := bBit5;
L_TBConvBitsToWord.6 := bBit6;
L_TBConvBitsToWord.7 := bBit7;
L_TBConvBitsToWord.8 := bBit8;
L_TBConvBitsToWord.9 := bBit9;
L_TBConvBitsToWord.10 := bBit10;
L_TBConvBitsToWord.11 := bBit11;
L_TBConvBitsToWord.12 := bBit12;
L_TBConvBitsToWord.13 := bBit13;
L_TBConvBitsToWord.14 := bBit14;
L_TBConvBitsToWord.15 := bBit15;

END_FUNCTION

// ---- POUs/Conversions/BitOriented/L_TBConvByteToBits.TcPOU
(****************************************************************************************)
(*							Beckhoff Automation Poland									*)
(*							L_TBConvByteToBits     v1.0									*)
(*									29.02.2007											*)
(*	This FB returns the 8 corresponding bit values for an input value of type ”byte”	*)
(*______________________________________________________________________________________*)
FUNCTION_BLOCK L_TBConvByteToBits
VAR_INPUT
	byInput: BYTE;
END_VAR
VAR_OUTPUT
	bBit0: BOOL;
	bBit1: BOOL;
	bBit2: BOOL;
	bBit3: BOOL;
	bBit4: BOOL;
	bBit5: BOOL;
	bBit6: BOOL;
	bBit7: BOOL;
END_VAR

bBit0 := byInput.0;
bBit1 := byInput.1;
bBit2 := byInput.2;
bBit3 := byInput.3;
bBit4 := byInput.4;
bBit5 := byInput.5;
bBit6 := byInput.6;
bBit7 := byInput.7;

END_FUNCTION_BLOCK

// ---- POUs/Conversions/BitOriented/L_TBConvDwordToArrBits.TcPOU
(****************************************************************************************)
(*							Beckhoff Automation Poland									*)
(*							L_TBConvDwordToArrBits v1.0									*)
(*									7.04.2009											*)
(* 				This F returns the 32 corresponding ARRAY of bit values 				*)
(*					for an input value of type ”double word”							*)
(*______________________________________________________________________________________*)
FUNCTION L_TBConvDwordToArrBits: ARRAY [0..31] OF BOOL
VAR_INPUT
	dwInput: DWORD;
END_VAR

L_TBConvDwordToArrBits[0]:=dwInput.0;
L_TBConvDwordToArrBits[1]:=dwInput.1;
L_TBConvDwordToArrBits[2]:=dwInput.2;
L_TBConvDwordToArrBits[3]:=dwInput.3;
L_TBConvDwordToArrBits[4]:=dwInput.4;
L_TBConvDwordToArrBits[5]:=dwInput.5;
L_TBConvDwordToArrBits[6]:=dwInput.6;
L_TBConvDwordToArrBits[7]:=dwInput.7;
L_TBConvDwordToArrBits[8]:=dwInput.8;
L_TBConvDwordToArrBits[9]:=dwInput.9;
L_TBConvDwordToArrBits[10]:=dwInput.10;
L_TBConvDwordToArrBits[11]:=dwInput.11;
L_TBConvDwordToArrBits[12]:=dwInput.12;
L_TBConvDwordToArrBits[13]:=dwInput.13;
L_TBConvDwordToArrBits[14]:=dwInput.14;
L_TBConvDwordToArrBits[15]:=dwInput.15;
L_TBConvDwordToArrBits[16]:=dwInput.16;
L_TBConvDwordToArrBits[17]:=dwInput.17;
L_TBConvDwordToArrBits[18]:=dwInput.18;
L_TBConvDwordToArrBits[19]:=dwInput.19;
L_TBConvDwordToArrBits[20]:=dwInput.20;
L_TBConvDwordToArrBits[21]:=dwInput.21;
L_TBConvDwordToArrBits[22]:=dwInput.22;
L_TBConvDwordToArrBits[23]:=dwInput.23;
L_TBConvDwordToArrBits[24]:=dwInput.24;
L_TBConvDwordToArrBits[25]:=dwInput.25;
L_TBConvDwordToArrBits[26]:=dwInput.26;
L_TBConvDwordToArrBits[27]:=dwInput.27;
L_TBConvDwordToArrBits[28]:=dwInput.28;
L_TBConvDwordToArrBits[29]:=dwInput.29;
L_TBConvDwordToArrBits[30]:=dwInput.30;
L_TBConvDwordToArrBits[31]:=dwInput.31;

END_FUNCTION

// ---- POUs/Conversions/BitOriented/L_TBConvDwordToBits.TcPOU
(****************************************************************************************)
(*							Beckhoff Automation Poland									*)
(*							L_TBConvDwordToBits v1.0									*)
(*									29.02.2007											*)
(* This FB returns the 32 corresponding bit values for an input value of type ”double word” *)
(*_______________________________________________________________________________________*)
FUNCTION_BLOCK L_TBConvDwordToBits
VAR_INPUT
	dwInput: DWORD;
END_VAR
VAR_OUTPUT
	bBit0: BOOL;
	bBit1: BOOL;
	bBit2: BOOL;
	bBit3: BOOL;
	bBit4: BOOL;
	bBit5: BOOL;
	bBit6: BOOL;
	bBit7: BOOL;
	bBit8: BOOL;
	bBit9: BOOL;
	bBit10: BOOL;
	bBit11: BOOL;
	bBit12: BOOL;
	bBit13: BOOL;
	bBit14: BOOL;
	bBit15: BOOL;
	bBit16: BOOL;
	bBit17: BOOL;
	bBit18: BOOL;
	bBit19: BOOL;
	bBit20: BOOL;
	bBit21: BOOL;
	bBit22: BOOL;
	bBit23: BOOL;
	bBit24: BOOL;
	bBit25: BOOL;
	bBit26: BOOL;
	bBit27: BOOL;
	bBit28: BOOL;
	bBit29: BOOL;
	bBit30: BOOL;
	bBit31: BOOL;
END_VAR
VAR
END_VAR

bBit0:=dwInput.0;
bBit1:=dwInput.1;
bBit2:=dwInput.2;
bBit3:=dwInput.3;
bBit4:=dwInput.4;
bBit5:=dwInput.5;
bBit6:=dwInput.6;
bBit7:=dwInput.7;
bBit8:=dwInput.8;
bBit9:=dwInput.9;
bBit10:=dwInput.10;
bBit11:=dwInput.11;
bBit12:=dwInput.12;
bBit13:=dwInput.13;
bBit14:=dwInput.14;
bBit15:=dwInput.15;
bBit16:=dwInput.16;
bBit17:=dwInput.17;
bBit18:=dwInput.18;
bBit19:=dwInput.19;
bBit20:=dwInput.20;
bBit21:=dwInput.21;
bBit22:=dwInput.22;
bBit23:=dwInput.23;
bBit24:=dwInput.24;
bBit25:=dwInput.25;
bBit26:=dwInput.26;
bBit27:=dwInput.27;
bBit28:=dwInput.28;
bBit29:=dwInput.29;
bBit30:=dwInput.30;
bBit31:=dwInput.31;

END_FUNCTION_BLOCK

// ---- POUs/Conversions/BitOriented/L_TBConvWordToBits.TcPOU
(****************************************************************************************)
(*							Beckhoff Automation Poland									*)
(*							L_TBConvWordToBits v1.0										*)
(*									29.02.2007											*)
(*	This FB returns the 16 corresponding bit values for an input value of type ” word”	*)
(*______________________________________________________________________________________*)
FUNCTION_BLOCK L_TBConvWordToBits
VAR_INPUT
	wInput:WORD;
END_VAR
VAR_OUTPUT
	bBit0: BOOL;
	bBit1: BOOL;
	bBit2: BOOL;
	bBit3: BOOL;
	bBit4: BOOL;
	bBit5: BOOL;
	bBit6: BOOL;
	bBit7: BOOL;
	bBit8: BOOL;
	bBit9: BOOL;
	bBit10: BOOL;
	bBit11: BOOL;
	bBit12: BOOL;
	bBit13: BOOL;
	bBit14: BOOL;
	bBit15: BOOL;
END_VAR
VAR
END_VAR

bBit0:=wInput.0;
bBit1:=wInput.1;
bBit2:=wInput.2;
bBit3:=wInput.3;
bBit4:=wInput.4;
bBit5:=wInput.5;
bBit6:=wInput.6;
bBit7:=wInput.7;
bBit8:=wInput.8;
bBit9:=wInput.9;
bBit10:=wInput.10;
bBit11:=wInput.11;
bBit12:=wInput.12;
bBit13:=wInput.13;
bBit14:=wInput.14;
bBit15:=wInput.15;

END_FUNCTION_BLOCK

// ---- POUs/Conversions/BitOriented/L_TBGetBitOfByte.TcPOU
(****************************************************************************************)
(*							Beckhoff Automation Poland									*)
(*								L_TBGetBitOfByte v1.0									*)
(*									29.02.2007											*)
(*				This function returns the state of a single bit within a ”byte” value	*)
(*______________________________________________________________________________________*)
FUNCTION L_TBGetBitOfByte : BOOL
VAR_INPUT
	byInput: BYTE;
	byBitNr: BYTE;
END_VAR

CASE byBitNr OF
	0:
	L_TBGetBitOfByte := byInput.0;
	1:
	L_TBGetBitOfByte := byInput.1;
	2:
	L_TBGetBitOfByte := byInput.2;
	3:
	L_TBGetBitOfByte := byInput.3;
	4:
	L_TBGetBitOfByte := byInput.4;
	5:
	L_TBGetBitOfByte := byInput.5;
	6:
	L_TBGetBitOfByte := byInput.6;
	7:
	L_TBGetBitOfByte := byInput.7;
END_CASE

END_FUNCTION

// ---- POUs/Conversions/BitOriented/L_TBGetBitOfDword.TcPOU
(****************************************************************************************)
(*							Beckhoff Automation Poland									*)
(*							L_TBGetBitOfDword v1.0										*)
(*									29.02.2007											*)
(*		This function returns the state of a single bit within a ”double word” value	*)
(*______________________________________________________________________________________*)
FUNCTION L_TBGetBitOfDword : BOOL
VAR_INPUT
	dwInput:DWORD;
	byBitNr:BYTE;
END_VAR
VAR
END_VAR

CASE byBitNr OF
	0:
	L_TBGetBitOfDword:=dwInput.0;
	1:
	L_TBGetBitOfDword:=dwInput.1;
	2:
	L_TBGetBitOfDword:=dwInput.2;
	3:
	L_TBGetBitOfDword:=dwInput.3;
	4:
	L_TBGetBitOfDword:=dwInput.4;
	5:
	L_TBGetBitOfDword:=dwInput.5;
	6:
	L_TBGetBitOfDword:=dwInput.6;
	7:
	L_TBGetBitOfDword:=dwInput.7;
	8:
	L_TBGetBitOfDword:=dwInput.8;
	9:
	L_TBGetBitOfDword:=dwInput.9;
	10:
	L_TBGetBitOfDword:=dwInput.10;
	11:
	L_TBGetBitOfDword:=dwInput.11;
	12:
	L_TBGetBitOfDword:=dwInput.12;
	13:
	L_TBGetBitOfDword:=dwInput.13;
	14:
	L_TBGetBitOfDword:=dwInput.14;
	15:
	L_TBGetBitOfDword:=dwInput.15;
	16:
	L_TBGetBitOfDword:=dwInput.16;
	17:
	L_TBGetBitOfDword:=dwInput.17;
	18:
	L_TBGetBitOfDword:=dwInput.18;
	19:
	L_TBGetBitOfDword:=dwInput.19;
	20:
	L_TBGetBitOfDword:=dwInput.20;
	21:
	L_TBGetBitOfDword:=dwInput.21;
	22:
	L_TBGetBitOfDword:=dwInput.22;
	23:
	L_TBGetBitOfDword:=dwInput.23;
	24:
	L_TBGetBitOfDword:=dwInput.24;
	25:
	L_TBGetBitOfDword:=dwInput.25;
	26:
	L_TBGetBitOfDword:=dwInput.26;
	27:
	L_TBGetBitOfDword:=dwInput.27;
	28:
	L_TBGetBitOfDword:=dwInput.28;
	29:
	L_TBGetBitOfDword:=dwInput.29;
	30:
	L_TBGetBitOfDword:=dwInput.30;
	31:
	L_TBGetBitOfDword:=dwInput.31;
END_CASE

END_FUNCTION

// ---- POUs/Conversions/BitOriented/L_TBGetBitOfWord.TcPOU
(****************************************************************************************)
(*							Beckhoff Automation Poland									*)
(*							L_TBGetBitOfWord v1.0										*)
(*									29.02.2007											*)
(*			This function returns the state of a single bit within a ”word” value		*)
(*______________________________________________________________________________________*)
FUNCTION L_TBGetBitOfWord : BOOL
VAR_INPUT
	wInput:WORD;
	byBitNr:BYTE;
END_VAR
VAR
END_VAR

CASE byBitNr OF
	0:
	L_TBGetBitOfWord:=wInput.0;
	1:
	L_TBGetBitOfWord:=wInput.1;
	2:
	L_TBGetBitOfWord:=wInput.2;
	3:
	L_TBGetBitOfWord:=wInput.3;
	4:
	L_TBGetBitOfWord:=wInput.4;
	5:
	L_TBGetBitOfWord:=wInput.5;
	6:
	L_TBGetBitOfWord:=wInput.6;
	7:
	L_TBGetBitOfWord:=wInput.7;
	8:
	L_TBGetBitOfWord:=wInput.8;
	9:
	L_TBGetBitOfWord:=wInput.9;
	10:
	L_TBGetBitOfWord:=wInput.10;
	11:
	L_TBGetBitOfWord:=wInput.11;
	12:
	L_TBGetBitOfWord:=wInput.12;
	13:
	L_TBGetBitOfWord:=wInput.13;
	14:
	L_TBGetBitOfWord:=wInput.14;
	15:
	L_TBGetBitOfWord:=wInput.15;
END_CASE

END_FUNCTION

// ---- POUs/Conversions/BitOriented/L_TBResetBitOfByte.TcPOU
(****************************************************************************************)
(*							Beckhoff Automation Poland									*)
(*							L_TBResetBitOfByte v1.0										*)
(*									29.02.2007											*)
(*				This function resets a single bit in a value of type ”byte” to “0”		*)
(*______________________________________________________________________________________*)
FUNCTION L_TBResetBitOfByte : BYTE
VAR_INPUT
	byInput: BYTE;
	byBitNr: BYTE;
END_VAR

L_TBResetBitOfByte := byInput;
CASE byBitNr OF
	0:
	L_TBResetBitOfByte.0 := FALSE;
	1:
	L_TBResetBitOfByte.1 := FALSE;
	2:
	L_TBResetBitOfByte.2 := FALSE;
	3:
	L_TBResetBitOfByte.3 := FALSE;
	4:
	L_TBResetBitOfByte.4 := FALSE;
	5:
	L_TBResetBitOfByte.5 := FALSE;
	6:
	L_TBResetBitOfByte.6 := FALSE;
	7:
	L_TBResetBitOfByte.7 := FALSE;
END_CASE

END_FUNCTION

// ---- POUs/Conversions/BitOriented/L_TBResetBitOfDword.TcPOU
(****************************************************************************************)
(*							Beckhoff Automation Poland									*)
(*							L_TBResetBitOfDword v1.0									*)
(*									29.02.2007											*)
(*			This function resets a single bit in a value of type ”double word” to “0”	*)
(*______________________________________________________________________________________*)
FUNCTION L_TBResetBitOfDword : DWORD
VAR_INPUT
	dwInput: DWORD;
	byBitNr: BYTE;
END_VAR
VAR
END_VAR

L_TBResetBitOfDword := dwInput;
CASE byBitNr OF
	0:
	L_TBResetBitOfDword.0 := FALSE;
	1:
	L_TBResetBitOfDword.1 := FALSE;
	2:
	L_TBResetBitOfDword.2 := FALSE;
	3:
	L_TBResetBitOfDword.3 := FALSE;
	4:
	L_TBResetBitOfDword.4 := FALSE;
	5:
	L_TBResetBitOfDword.5 := FALSE;
	6:
	L_TBResetBitOfDword.6 := FALSE;
	7:
	L_TBResetBitOfDword.7 := FALSE;
	8:
	L_TBResetBitOfDword.8 := FALSE;
	9:
	L_TBResetBitOfDword.9 := FALSE;
	10:
	L_TBResetBitOfDword.10 := FALSE;
	11:
	L_TBResetBitOfDword.11 := FALSE;
	12:
	L_TBResetBitOfDword.12 := FALSE;
	13:
	L_TBResetBitOfDword.13 := FALSE;
	14:
	L_TBResetBitOfDword.14 := FALSE;
	15:
	L_TBResetBitOfDword.15 := FALSE;
	16:
	L_TBResetBitOfDword.16 := FALSE;
	17:
	L_TBResetBitOfDword.17 := FALSE;
	18:
	L_TBResetBitOfDword.18 := FALSE;
	19:
	L_TBResetBitOfDword.19 := FALSE;
	20:
	L_TBResetBitOfDword.20 := FALSE;
	21:
	L_TBResetBitOfDword.21 := FALSE;
	22:
	L_TBResetBitOfDword.22 := FALSE;
	23:
	L_TBResetBitOfDword.23 := FALSE;
	24:
	L_TBResetBitOfDword.24 := FALSE;
	25:
	L_TBResetBitOfDword.25 := FALSE;
	26:
	L_TBResetBitOfDword.26 := FALSE;
	27:
	L_TBResetBitOfDword.27 := FALSE;
	28:
	L_TBResetBitOfDword.28 := FALSE;
	29:
	L_TBResetBitOfDword.29 := FALSE;
	30:
	L_TBResetBitOfDword.30 := FALSE;
	31:
	L_TBResetBitOfDword.31 := FALSE;
END_CASE

END_FUNCTION

// ---- POUs/Conversions/BitOriented/L_TBResetBitOfWord.TcPOU
(****************************************************************************************)
(*							Beckhoff Automation Poland									*)
(*							L_TBResetBitOfWord v1.0										*)
(*									29.02.2007											*)
(*				This function resets a single bit in a value of type ”word” to “0”		*)
(*______________________________________________________________________________________*)
FUNCTION L_TBResetBitOfWord : WORD
VAR_INPUT
	wInput: WORD;
	byBitNr: BYTE;
END_VAR
VAR
END_VAR

L_TBResetBitOfWord := wInput;
CASE byBitNr OF
	0:
	L_TBResetBitOfWord.0 := FALSE;
	1:
	L_TBResetBitOfWord.1 := FALSE;
	2:
	L_TBResetBitOfWord.2 := FALSE;
	3:
	L_TBResetBitOfWord.3 := FALSE;
	4:
	L_TBResetBitOfWord.4 := FALSE;
	5:
	L_TBResetBitOfWord.5 := FALSE;
	6:
	L_TBResetBitOfWord.6 := FALSE;
	7:
	L_TBResetBitOfWord.7 := FALSE;
	8:
	L_TBResetBitOfWord.8 := FALSE;
	9:
	L_TBResetBitOfWord.9 := FALSE;
	10:
	L_TBResetBitOfWord.10 := FALSE;
	11:
	L_TBResetBitOfWord.11 := FALSE;
	12:
	L_TBResetBitOfWord.12 := FALSE;
	13:
	L_TBResetBitOfWord.13 := FALSE;
	14:
	L_TBResetBitOfWord.14 := FALSE;
	15:
	L_TBResetBitOfWord.15 := FALSE;
END_CASE

END_FUNCTION

// ---- POUs/Conversions/BitOriented/L_TBSetBitOfByte.TcPOU
(****************************************************************************************)
(*							Beckhoff Automation Poland									*)
(*							L_TBSetBitOfByte v1.0										*)
(*									29.02.2007											*)
(*				This function sets a single bit in a value of type ”byte” to “1”		*)
(*______________________________________________________________________________________*)
FUNCTION L_TBSetBitOfByte : BYTE
VAR_INPUT
	byInput: BYTE;
	byBitNr: BYTE;
END_VAR

L_TBSetBitOfByte := byInput;
CASE byBitNr OF
	0:
	L_TBSetBitOfByte.0 := TRUE;
	1:
	L_TBSetBitOfByte.1 := TRUE;
	2:
	L_TBSetBitOfByte.2 := TRUE;
	3:
	L_TBSetBitOfByte.3 := TRUE;
	4:
	L_TBSetBitOfByte.4 := TRUE;
	5:
	L_TBSetBitOfByte.5 := TRUE;
	6:
	L_TBSetBitOfByte.6 := TRUE;
	7:
	L_TBSetBitOfByte.7 := TRUE;
END_CASE

END_FUNCTION

// ---- POUs/Conversions/BitOriented/L_TBSetBitOfDword.TcPOU
(****************************************************************************************)
(*							Beckhoff Automation Poland									*)
(*							L_TBSetBitOfDword v1.0										*)
(*									29.02.2007											*)
(*			This function sets a single bit in a value of type ”double word” to “1”		*)
(*______________________________________________________________________________________*)
FUNCTION L_TBSetBitOfDword : DWORD
VAR_INPUT
	dwInput: DWORD;
	byBitNr: BYTE;
END_VAR
VAR
END_VAR

L_TBSetBitOfDword := dwInput;
CASE byBitNr OF
	0:
	L_TBSetBitOfDword.0 := TRUE;
	1:
	L_TBSetBitOfDword.1 := TRUE;
	2:
	L_TBSetBitOfDword.2 := TRUE;
	3:
	L_TBSetBitOfDword.3 := TRUE;
	4:
	L_TBSetBitOfDword.4 := TRUE;
	5:
	L_TBSetBitOfDword.5 := TRUE;
	6:
	L_TBSetBitOfDword.6 := TRUE;
	7:
	L_TBSetBitOfDword.7 := TRUE;
	8:
	L_TBSetBitOfDword.8 := TRUE;
	9:
	L_TBSetBitOfDword.9 := TRUE;
	10:
	L_TBSetBitOfDword.10 := TRUE;
	11:
	L_TBSetBitOfDword.11 := TRUE;
	12:
	L_TBSetBitOfDword.12 := TRUE;
	13:
	L_TBSetBitOfDword.13 := TRUE;
	14:
	L_TBSetBitOfDword.14 := TRUE;
	15:
	L_TBSetBitOfDword.15 := TRUE;
	16:
	L_TBSetBitOfDword.16 := TRUE;
	17:
	L_TBSetBitOfDword.17 := TRUE;
	18:
	L_TBSetBitOfDword.18 := TRUE;
	19:
	L_TBSetBitOfDword.19 := TRUE;
	20:
	L_TBSetBitOfDword.20 := TRUE;
	21:
	L_TBSetBitOfDword.21 := TRUE;
	22:
	L_TBSetBitOfDword.22 := TRUE;
	23:
	L_TBSetBitOfDword.23 := TRUE;
	24:
	L_TBSetBitOfDword.24 := TRUE;
	25:
	L_TBSetBitOfDword.25 := TRUE;
	26:
	L_TBSetBitOfDword.26 := TRUE;
	27:
	L_TBSetBitOfDword.27 := TRUE;
	28:
	L_TBSetBitOfDword.28 := TRUE;
	29:
	L_TBSetBitOfDword.29 := TRUE;
	30:
	L_TBSetBitOfDword.30 := TRUE;
	31:
	L_TBSetBitOfDword.31 := TRUE;
END_CASE

END_FUNCTION

// ---- POUs/Conversions/BitOriented/L_TBSetBitOfWord.TcPOU
(****************************************************************************************)
(*							Beckhoff Automation Poland									*)
(*							L_TBSetBitOfWord v1.0										*)
(*									29.02.2007											*)
(*				This function sets a single bit in a value of type ”word” to “1”		*)
(*______________________________________________________________________________________*)
FUNCTION L_TBSetBitOfWord : WORD
VAR_INPUT
	wInput: WORD;
	byBitNr: BYTE;
END_VAR
VAR
END_VAR

L_TBSetBitOfWord := wInput;
CASE byBitNr OF
	0:
	L_TBSetBitOfWord.0 := TRUE;
	1:
	L_TBSetBitOfWord.1 := TRUE;
	2:
	L_TBSetBitOfWord.2 := TRUE;
	3:
	L_TBSetBitOfWord.3 := TRUE;
	4:
	L_TBSetBitOfWord.4 := TRUE;
	5:
	L_TBSetBitOfWord.5 := TRUE;
	6:
	L_TBSetBitOfWord.6 := TRUE;
	7:
	L_TBSetBitOfWord.7 := TRUE;
	8:
	L_TBSetBitOfWord.8 := TRUE;
	9:
	L_TBSetBitOfWord.9 := TRUE;
	10:
	L_TBSetBitOfWord.10 := TRUE;
	11:
	L_TBSetBitOfWord.11 := TRUE;
	12:
	L_TBSetBitOfWord.12 := TRUE;
	13:
	L_TBSetBitOfWord.13 := TRUE;
	14:
	L_TBSetBitOfWord.14 := TRUE;
	15:
	L_TBSetBitOfWord.15 := TRUE;
END_CASE

END_FUNCTION

// ---- POUs/Conversions/BitOriented/L_TBSquareWave.TcPOU
(****************************************************************************************)
(*							Beckhoff Automation Poland									*)
(*								L_TBSquareWave v1.0										*)
(*									29.02.2007											*)
(*	This FB can be used to generate a Boolean square wave signal with a variable high/low time *)
(*______________________________________________________________________________________*)
FUNCTION_BLOCK L_TBSquareWave
VAR_INPUT
	bEnable:BOOL;
	wTimeHigh:WORD;
	wTimeLow:WORD;
END_VAR
VAR_OUTPUT
	bOut:BOOL;
END_VAR
VAR
	ton1: TON;
	ton2: TON;
END_VAR

IF bEnable THEN
	ton1(IN:= NOT ton2.Q, PT:=WORD_TO_TIME(wTimeLow));
	bOut:=NOT ton1.Q;
	ton2(IN:=ton1.Q , PT:=WORD_TO_TIME(wTimeHigh));
ELSE
	bOut:=FALSE;
END_IF

END_FUNCTION_BLOCK

// ---- POUs/Conversions/FB_CONCAT_S2040.TcPOU
(****************************************************************************************)
(*							Beckhoff Automation Poland									*)
(*							FB_CONCAT_S2040	 v1.0										*)
(*									24.5.2011											*)
(*				Blok funkcyjny łączący do 8 zmiennych trypu STRING(max 255 znaków)		*)
(*						w jedną zmienną typu ST_STRING_2040								*)
(*______________________________________________________________________________________*)
FUNCTION_BLOCK FB_CONCAT_S2040
VAR_INPUT
	sString1								:	STRING(255);
END_VAR
VAR
	i										:	INT;				(*iterator*)
	k										:	INT;				(*ostatni zaczety string*)
	wLength									:	WORD;				(*dlugosc ostatniego STRINGa*)
END_VAR
VAR_IN_OUT
	VeryLongString							:	ST_STRING_2040;
END_VAR
VAR_OUTPUT
	wIloscWszystkichZnakow					:	WORD;
END_VAR

k:=0;
wLength:=0;
FOR i := 1 TO 8 DO
	IF LEN(VeryLongString[i]) <> 0 THEN
		wLength := INT_TO_WORD(LEN(VeryLongString[i]));
		k := i;
	END_IF
END_FOR
(* Nie bylo jeszce nic wpisane *)
IF k = 0 THEN
	wIloscWszystkichZnakow := INT_TO_WORD(LEN(sString1));
	MEMCPY(ADR(VeryLongString), ADR(sString1), INT_TO_UINT(LEN(sString1)));
ELSE
	wIloscWszystkichZnakow := INT_TO_WORD((k-1)*256+WORD_TO_INT(wLength));
	IF (WORD_TO_INT(wIloscWszystkichZnakow)+LEN(sString1)) > 2047 THEN
		MEMCPY(ADR(VeryLongString)+wIloscWszystkichZnakow, ADR(sString1), 2047 - wIloscWszystkichZnakow );
	ELSE
		MEMCPY(ADR(VeryLongString)+wIloscWszystkichZnakow, ADR(sString1), INT_TO_UINT(LEN(sString1)));
	END_IF
	wIloscWszystkichZnakow := int_to_word(word_to_int(wIloscWszystkichZnakow) + LEN(sString1));
END_IF

END_FUNCTION_BLOCK

// ---- POUs/Conversions/FB_IntTo2Byte.TcPOU
(****************************************************************************************)
(*							Beckhoff Automation Poland									*)
(*								FB_IntTo2Byte	 v1.0									*)
(*									24.5.2011											*)
(*			Blok funkcyjny rozbijający zmienną typu INT na dwie zmienne typu BYTE		*)
(*______________________________________________________________________________________*)
FUNCTION_BLOCK FB_IntTo2Byte
VAR_INPUT
	iInput :INT;
END_VAR
VAR_OUTPUT
	byStarszy : BYTE;
	byMlodszy : BYTE;
END_VAR

byMlodszy := INT_TO_BYTE(iInput);
byStarszy := INT_TO_BYTE(ROL(iInput, 8));

END_FUNCTION_BLOCK

// ---- POUs/Conversions/F_4BYTES_TO_DWORD.TcPOU
(****************************************************************************)
(*							Beckhoff Automation Poland						*)
(*							F_4BYTES_TO_DWORD v1							*)
(*									21.11.2013								*)
(*					Funkcja zamieniająca 4 zmienne typu BYTE na DWORD 		*)
(*__________________________________________________________________________*)
FUNCTION F_4BYTES_TO_DWORD : DWORD
VAR_INPUT
	BByte0		: BYTE;
	BByte1		: BYTE;
	BByte2		: BYTE;
	BByte3		: BYTE;
END_VAR

F_4BYTES_TO_DWORD := BByte3 *16#1000000 + BByte2 *16#10000 + BByte1 *16#100 + BByte0;

END_FUNCTION

// ---- POUs/Conversions/F_4BYTES_TO_REAL.TcPOU
(************************************************************************************)
(*							Beckhoff Automation Poland								*)
(*							F_4BYTES_TO_REAL v1										*)
(*									21.11.2013										*)
(*					Funkcja zamieniająca 4 zmienne typu BYTE na REAL	 			*)
(*__________________________________________________________________________________*)
FUNCTION F_4BYTES_TO_REAL : REAL
VAR_INPUT
	BByte0		: BYTE;
	BByte1		: BYTE;
	BByte2		: BYTE;
	BByte3		: BYTE;
END_VAR
VAR
	dwDword	: DWORD;
END_VAR

dwDword := BByte3 *16#1000000 + BByte2 *16#10000 + BByte1 *16#100 + BByte0;
MEMCPY(ADR(F_4BYTES_TO_REAL),ADR(dwDword), 4);

END_FUNCTION

// ---- POUs/Conversions/F_8BYTES_TO_LREAL.TcPOU
(************************************************************************************)
(*							Beckhoff Automation Poland								*)
(*							F_8BYTES_TO_LREAL v1.0									*)
(*									3.07.2015										*)
(*					Funkcja zamieniająca 8 zmiennych typu BYTE na LREAL 			*)
(*__________________________________________________________________________________*)
FUNCTION F_8BYTES_TO_LREAL : LREAL
VAR_INPUT
	BByte0		: BYTE;
	BByte1		: BYTE;
	BByte2		: BYTE;
	BByte3		: BYTE;
	BByte4		: BYTE;
	BByte5		: BYTE;
	BByte6		: BYTE;
	BByte7		: BYTE;
END_VAR
VAR
	arrByte	: ARRAY [1..8] OF BYTE;
END_VAR

arrByte[1] := BByte0;
arrByte[2] := BByte1;
arrByte[3] := BByte2;
arrByte[4] := BByte3;
arrByte[5] := BByte4;
arrByte[6] := BByte5;
arrByte[7] := BByte6;
arrByte[8] := BByte7;

MEMCPY(ADR(F_8BYTES_TO_LREAL),ADR(arrByte), 8);

END_FUNCTION

// ---- POUs/Conversions/F_BCDToDec.TcPOU
(************************************************************************************)
(*								Beckhoff Automation Poland							*)
(* 									F_BCDToDec v1.0									*)
(* 										26.06.2014									*)
(*					Funkcja konwertujaca BYTE (kod BCD) na BYTE (DEC)				*)
(*__________________________________________________________________________________*)
FUNCTION F_BCDToDec: BYTE
VAR_INPUT
	BIn:BYTE;
END_VAR

CASE ROL(BIn AND 16#F0,4) OF
0:	F_BCDToDec := 00;
1:	F_BCDToDec := 10;
2:	F_BCDToDec := 20;
3:	F_BCDToDec := 30;
4:	F_BCDToDec := 40;
5:	F_BCDToDec := 50;
6:	F_BCDToDec := 60;
7:	F_BCDToDec := 70;
8:	F_BCDToDec := 80;
9:	F_BCDToDec := 90;
ELSE
	;
END_CASE

CASE BIn AND 16#F OF
0..9:	F_BCDToDec := F_BCDToDec + (BIn AND 16#F);
ELSE
	;
END_CASE

END_FUNCTION

// ---- POUs/Conversions/F_CLEAN_S2040.TcPOU
(****************************************************************************************)
(*							Beckhoff Automation Poland									*)
(*								F_CLEAN_S2040	 v1.0									*)
(*									24.5.2011											*)
(*				Funkcja czyszcząca zawartość zmiennej typu ST_STRING_2040				*)
(*______________________________________________________________________________________*)
FUNCTION F_CLEAN_S2040 : ST_STRING_2040
VAR_INPUT
                VeryLongString: ST_STRING_2040;
END_VAR
VAR
                i: INT;                    (*iterator*)
END_VAR

FOR i := 1 TO 8 DO
                VeryLongString[i] := '$N';
END_FOR

END_FUNCTION

// ---- POUs/Conversions/F_Convert_4BBCD_To_Real.TcPOU
(************************************************************************************************)
(*								Beckhoff Automation Poland										*)
(* 									F_Convert_4BBCD_To_Real v1.0								*)
(* 										26.06.2014												*)
(*	Funkcja konwertujaca 4 zmienne typu BYTE (BCD) na REAL - czesto spotykane w protokole M-Bus	*)
(*______________________________________________________________________________________________*)
FUNCTION F_Convert_4BBCD_To_Real : REAL
VAR_INPUT
	Byte1: BYTE; (* LSB *)
	Byte2: BYTE;
	Byte3: BYTE;
	Byte4: BYTE; (* MSB *)
END_VAR

F_Convert_4BBCD_To_Real := udint_to_real(F_BCDToDec(Byte1)*1+F_BCDToDec(Byte2)*100+F_BCDToDec(Byte3)*10000+F_BCDToDec(Byte4)*1000000);

END_FUNCTION

// ---- POUs/Conversions/F_DWORD_TO_REAL.TcPOU
(********************************************************************************)
(*							Beckhoff Automation Poland							*)
(*							F_DWORD_TO_REAL v1									*)
(*									21.11.2013									*)
(*					Funkcja zamieniająca DWORD na REAL				 			*)
(*______________________________________________________________________________*)
FUNCTION F_DWORD_TO_REAL : REAL
VAR_INPUT
	dwDword	: DWORD;
END_VAR

MEMCPY(ADR(F_DWORD_TO_REAL),ADR(dwDword), 4);

END_FUNCTION

// ---- POUs/Conversions/F_Words_to_Real.TcPOU
(********************************************************************************************)
(*							Beckhoff Automation Poland										*)
(*							F_Words_to_Real													*)
(*									12.05.2011												*)
(*			Funkcja składa dwie wartości typu WORD  i zamienia na watrosc typu REAL			*)
(*__________________________________________________________________________________________*)

FUNCTION F_Words_to_Real : REAL
VAR_INPUT
	wUpperWord : WORD;
	wLowerWord :WORD;
END_VAR
VAR
END_VAR

MEMCPY(ADR(F_Words_to_Real),ADR(wUpperWord),2);
MEMCPY(ADR(F_Words_to_Real)+2,ADR(wLowerWord),2);

END_FUNCTION

// ---- POUs/Conversions/GRAYB_TO_WORD.TcPOU
(****************************************************************************************)
(*							Beckhoff Automation Poland									*)
(*							GRAYB_TO_WORD	 v1.0										*)
(*									29.12.2008											*)
(*		Funkcja konwerująca 16 sygnalow typu BOOL tworzacych kod Graya					*)
(*						 na wartosc decymalna typu WORD									*)
(*______________________________________________________________________________________*)
FUNCTION GRAYB_TO_WORD : WORD
VAR_INPUT
	bIn0: BOOL;
	bIn1: BOOL;
	bIn2: BOOL;
	bIn3: BOOL;
	bIn4: BOOL;
	bIn5: BOOL;
	bIn6: BOOL;
	bIn7: BOOL;
	bIn8: BOOL;
	bIn9: BOOL;
	bIn10: BOOL;
	bIn11: BOOL;
	bIn12: BOOL;
	bIn13: BOOL;
	bIn14: BOOL;
	bIn15: BOOL;
END_VAR

GRAYB_TO_WORD.15 := bIn15 XOR 0;
GRAYB_TO_WORD.14 := bIn14 XOR GRAYB_TO_WORD.15;
GRAYB_TO_WORD.13 := bIn13 XOR GRAYB_TO_WORD.14;
GRAYB_TO_WORD.12 := bIn12 XOR GRAYB_TO_WORD.13;
GRAYB_TO_WORD.11 := bIn11 XOR GRAYB_TO_WORD.12;
GRAYB_TO_WORD.10 := bIn10 XOR GRAYB_TO_WORD.11;
GRAYB_TO_WORD.9 := bIn9 XOR GRAYB_TO_WORD.10;
GRAYB_TO_WORD.8 := bIn8 XOR GRAYB_TO_WORD.9;
GRAYB_TO_WORD.7 := bIn7 XOR GRAYB_TO_WORD.8;
GRAYB_TO_WORD.6 := bIn6 XOR GRAYB_TO_WORD.7;
GRAYB_TO_WORD.5 := bIn5 XOR GRAYB_TO_WORD.6;
GRAYB_TO_WORD.4 := bIn4 XOR GRAYB_TO_WORD.5;
GRAYB_TO_WORD.3 := bIn3 XOR GRAYB_TO_WORD.4;
GRAYB_TO_WORD.2 := bIn2 XOR GRAYB_TO_WORD.3;
GRAYB_TO_WORD.1 := bIn1 XOR GRAYB_TO_WORD.2;
GRAYB_TO_WORD.0 := bIn0 XOR GRAYB_TO_WORD.1;

END_FUNCTION

// ---- POUs/Conversions/GRAYW_TO_WORD.TcPOU
(****************************************************************************************)
(*							Beckhoff Automation Poland									*)
(*							GRAYW_TO_WORD	 v1.0										*)
(*									29.12.2008											*)
(*		Funkcja konwerująca wartosc wejsciowa typu WORD zapisana w kodzie Graya			*)
(*						 na wartosc decymalna typu WORD									*)
(*______________________________________________________________________________________*)
FUNCTION GRAYW_TO_WORD : WORD
VAR_INPUT
	wIn:WORD;
END_VAR
VAR
END_VAR

GRAYW_TO_WORD.15 := wIn.15 XOR 0;
GRAYW_TO_WORD.14 := wIn.14 XOR GRAYW_TO_WORD.15;
GRAYW_TO_WORD.13 := wIn.13 XOR GRAYW_TO_WORD.14;
GRAYW_TO_WORD.12 := wIn.12 XOR GRAYW_TO_WORD.13;
GRAYW_TO_WORD.11 := wIn.11 XOR GRAYW_TO_WORD.12;
GRAYW_TO_WORD.10 := wIn.10 XOR GRAYW_TO_WORD.11;
GRAYW_TO_WORD.9 := wIn.9 XOR GRAYW_TO_WORD.10;
GRAYW_TO_WORD.8 := wIn.8 XOR GRAYW_TO_WORD.9;
GRAYW_TO_WORD.7 := wIn.7 XOR GRAYW_TO_WORD.8;
GRAYW_TO_WORD.6 := wIn.6 XOR GRAYW_TO_WORD.7;
GRAYW_TO_WORD.5 := wIn.5 XOR GRAYW_TO_WORD.6;
GRAYW_TO_WORD.4 := wIn.4 XOR GRAYW_TO_WORD.5;
GRAYW_TO_WORD.3 := wIn.3 XOR GRAYW_TO_WORD.4;
GRAYW_TO_WORD.2 := wIn.2 XOR GRAYW_TO_WORD.3;
GRAYW_TO_WORD.1 := wIn.1 XOR GRAYW_TO_WORD.2;
GRAYW_TO_WORD.0 := wIn.0 XOR GRAYW_TO_WORD.1;

END_FUNCTION

// ---- POUs/DateAndTime/FB_AstrTimeCET.TcPOU
(****************************************************************************************************)
(*							Beckhoff Automation Poland												*)
(*								FB_AstrTimeCET v1.0													*)
(*									24.10.2014														*)
(*	Blok funkcyjny zegara astronomicznego -  załączający wyjście bOutCET gdy jest dzien				*)
(*	 mozliwe jest wprowadzenie offsetu, który jest uwzgledniony przez wyjscie bOutCETOffs			*)
(*				Wymaga podania aktualnego czasu, informacji czy jest czas letni						*)
(* 			oraz szerokości rWidth i długości rLenght geograficznej obiektu							*)
(*					(w formie zmiennej typu REAL - 51 st 45 min = 51.75 !! )						*)
(*		Na wyjsciu podany jest również czas wschodu i zachodu Słońca w danym dniu					*)
(*					Wymagane dodanie biblioteki TcMatch 				 							*)
(*__________________________________________________________________________________________________*)
FUNCTION_BLOCK FB_AstrTimeCET
VAR_INPUT
	bCalculate				: BOOL;									(* Obliczenia na zadanie na obliczenia*)
	stActTimeCET			: TIMESTRUCT;							(* Aktualny czas CET*)
	rWidth					: REAL			:=52.059625;			(* szerokosc geograficzna ujemna - S  dodatnia - N, wspolrzedne Warszawy: 52° N; 21° E *)
	rLenght					: REAL			:=21.04540559999998;	(* dlugosc geograficzna ujemna - W  dodatnia - E*)
	bDSTSummer				: BOOL;									(* Sygnalizacja czasu letniego - GMT + 1h *)
	iSunriseOffset			: INT; 									(* przesuniecie zalaczenia, w minutach, "-" - wcześniej*)
	iSunsetOffset			: INT;									(* przesuniecie wylaczenia, w minutach, "-" - wcześniej*)
END_VAR
VAR_OUTPUT
	bOutCET					: BOOL;									(* Wskazanie dnia, TRUE => dzien, FALSE => noc*)
	bOutCETOffs				: BOOL; 								(* Wyjscie uwzgledniajace offset, TRUE => dzien, FALSE => noc*)
	todSunriseCET			: TOD;
	todSunsetCET			: TOD;
	todSunriseCETOffs		: TOD;
	todSunsetCETOffs		: TOD;
	bError					: BOOL; 								(* Blad nie podano czasu *)
END_VAR
VAR
	J,Cent,L,G,O,F,E,A,C,lrWsch,lrZach:	LREAL;
	wDayOld					: WORD;
	todSunriseGMT			: TOD;
	todSunsetGMT			: TOD;
	dwSunriseHourGMT		: DWORD;		(*Czas GMT wschodu i zachodu Słońca *)
	dwSunriseMinuteGMT		: DWORD;
	dwSunsetHourGMT			: DWORD;
	dwSunsetMinuteGMT		: DWORD;
	dwSunriseGMT			: DWORD;		(*czas wschodu GMT w ms*)
	dwSunsetGMT				: DWORD;		(*czas zachodu GMT w ms*)
	dwSunriseCET			: DWORD;		(*czas wschodu CET w ms*)
	dwSunsetCET				: DWORD;		(*czas zachodu CET w ms*)
	dwSunriseOffs			: DWORD;		(*czas wschodu CET z Offs w ms*)
	dwSunsetOffs			: DWORD;		(*czas zachodu CET z Offs w ms*)
	todActTime				: TOD;
END_VAR
VAR CONSTANT
	Req						: REAL := -0.833;		(*wysokosc Slonca podczas Wschodu i Zachodu*)
(*
Req = -0.833 - dla wschodów i zachodów Słońca
Req = -6 - dla zmierzchu cywilnego
Req = -12 - dla zmierzchu żeglarskiego
Req = -18 - dla zmierzchu astronomicznego
*)
END_VAR

bError := stActTimeCET.wYear = 0;
(*Obliczenia wykonywane sa gdy pobrany zostal czas po wykryciu nowego dnia lub na zadanie *)
IF NOT bError AND (bCalculate OR stActTimeCET.wDay <> wDayOld) THEN
	(*Bardzo skomplikowane obliczenia wschodu i zachod słońca dla czasu GMT*)
	J:=367*stActTimeCET.wYear-TRUNC(7*(stActTimeCET.wYear+TRUNC((stActTimeCET.wMonth+9)/12))/4)+TRUNC(275*stActTimeCET.wMonth/9)+stActTimeCET.wDay-730531.5;
	Cent:=J/36525;
	L:= LMOD((4.8949504201433+628.331969753199*Cent),6.28318530718);
	G:= LMOD((6.2400408+628.3019501*Cent),6.28318530718);
	O:=0.409093-0.0002269*Cent;
	F:=0.033423*SIN(G)+0.00034907*SIN(2*G);
	E:=0.0430398*SIN(2*(L+F)) - 0.00092502*SIN(4*(L+F)) - F;
	A:=ASIN(SIN(O)*SIN(L+F));
	C:=(SIN(0.017453293*Req) - SIN(0.017453293*rWidth)*SIN(A))/(COS(0.017453293*rWidth)*COS(A));
	lrWsch:=((PI - (E+0.017453293*rLenght + 1*ACOS(C)))*57.29577951/15);
	lrZach:=((PI - (E+0.017453293*rLenght + -1*ACOS(C)))*57.29577951/15);

	(*Obliczenie zmiennych dla czasu GMT*)
	dwSunriseHourGMT 	:= DINT_TO_DWORD(TRUNC(lrWsch));
	dwSunriseMinuteGMT 	:= LREAL_TO_DWORD((lrWsch - DWORD_TO_LREAL(dwSunriseHourGMT))*60);
	dwSunsetHourGMT 		:= DINT_TO_DWORD(TRUNC(lrZach));
	dwSunsetMinuteGMT 	:= LREAL_TO_DWORD((lrZach - DWORD_TO_LREAL(dwSunsetHourGMT))*60);
	dwSunriseGMT			:= (dwSunriseHourGMT*60+dwSunriseMinuteGMT)*60000;
	dwSunsetGMT			:= (dwSunsetHourGMT*60+dwSunsetMinuteGMT)*60000;
	todSunriseGMT 			:= DWORD_TO_TOD(dwSunriseGMT);
	todSunsetGMT 			:= DWORD_TO_TOD(dwSunsetGMT);

	(*Obliczenie zmiennych dla czasu CET*)
	dwSunriseCET 			:= dwSunriseGMT+3600000;
	dwSunsetCET			:= dwSunsetGMT+3600000;
	(* + 1h dla DST *)
	IF bDSTSummer THEN
		dwSunriseCET 		:= dwSunriseCET+3600000;
		dwSunsetCET		:= dwSunsetCET+3600000;
	END_IF
	todSunriseCET 			:= DWORD_TO_TOD(dwSunriseCET);
	todSunsetCET 			:= DWORD_TO_TOD(dwSunsetCET);

	(*Obliczenie zmiennych dla czasu CET z offsetem*)
	dwSunriseOffs 			:= dwSunriseCET + INT_TO_DWORD(iSunriseOffset)*60000;
	dwSunriseOffs 			:= LIMIT(0, dwSunriseOffs,86400000);						(* Jesli ktos przesadzil z offsetem i wyszedl poza dobe, to ustawiamy gorny limit *)
	dwSunsetOffs 			:= dwSunsetCET + INT_TO_DWORD(iSunsetOffset)*60000;
	dwSunsetOffs 			:= LIMIT(dwSunriseOffs, dwSunsetOffs,86400000);			(* Jesli ktos przesadzil z offsetem i wyszedl poza dobe, to ustawiamy gorny limit *)
	todSunriseCETOffs 		:= DWORD_TO_TOD(dwSunriseOffs);
	todSunsetCETOffs 		:= DWORD_TO_TOD(dwSunsetOffs);

	wDayOld 				:= stActTimeCET.wDay; (*ustawienie nowego dnia*)
END_IF
todActTime 					:= DT_TO_TOD(SYSTEMTIME_TO_DT(stActTimeCET));
(* Wystawienie wyjsc tylko gdy nie ma bledu*)
bOutCET 					:= NOT bError AND (todActTime >= todSunriseCET AND todActTime <= todSunsetCET);
bOutCETOffs 				:= NOT bError AND (todActTime >= todSunriseCETOffs AND todActTime <= todSunsetCETOffs);

END_FUNCTION_BLOCK

// ---- POUs/DateAndTime/FB_CycleTime.TcPOU
(************************************************************************************************)
(*								Beckhoff Automation Poland										*)
(* 									FB_CycleTime v1.0											*)
(* 										2.2.2011												*)
(*Blok funkcyjny podający na wyjściu czas miedzy kolejnymi wywołaniami - najczęściej czas cyklu	*)
(*______________________________________________________________________________________________*)
FUNCTION_BLOCK FB_CycleTime
VAR_INPUT
	bEnable		: 	BOOL:=TRUE; (* Zezwolenie na obliczenia *)
END_VAR
VAR_OUTPUT
	tCycleTime	:	TIME; 		(* Czas cylku *)
END_VAR
VAR
	x 			:	TIME;
	y 			:	TIME;
END_VAR

IF bEnable THEN
	x := TIME();
	tCycleTime := x-y;
	y:=x;
END_IF

END_FUNCTION_BLOCK

// ---- POUs/DateAndTime/FB_DST.TcPOU
(****************************************************************************************************)
(*							Beckhoff Automation Poland												*)
(*									FB_DST v 1.0													*)
(*									24.10.2014														*)
(*		Blok funkcyjny sprawdzajacy czy jest czas letni i obliczajacy czas lokalny CET z GMT		*)
(*					Działa w latach 2011 - 2030, poza tym zakresem podaje błąd						*)
(* 			Jesli chcemy obliczyc czas CET to wejsciu powienien być podany aktualny czas GMT		*)
(*__________________________________________________________________________________________________*)
FUNCTION_BLOCK FB_DST
VAR_INPUT
	dtActualTimeGMT: 	DT; 				(* Aktulany czas GMT*)
END_VAR
VAR_OUTPUT
	bSummerTime: 		BOOL;				(* TRUE gdy czas letni *)
	dtActualTimeCET: 	DT; 				(* Aktulany czas CET*)
	bError: 			BOOL;				(* TRUE jeśli podano nieprawidłowy rok *)
END_VAR
VAR
	dwActualTime: 		DWORD;
	dwYear: 			DWORD;
	t1: 				TON;
END_VAR
VAR CONSTANT
	(* Tablice z datami zmiany czasu *)
	aMarch:		ARRAY [2011..2030] OF DT := 	[DT#2011-03-27-01:00,DT#2012-03-25-01:00,DT#2013-03-31-01:00,DT#2014-03-30-01:00,DT#2015-03-29-01:00,
											DT#2016-03-27-01:00,DT#2017-03-26-01:00,DT#2018-03-25-01:00,DT#2019-03-31-01:00,DT#2020-03-29-01:00,
											DT#2021-03-28-01:00,DT#2022-03-27-01:00,DT#2023-03-26-01:00,DT#2024-03-31-01:00,DT#2025-03-30-01:00,
											DT#2026-03-29-01:00,DT#2027-03-28-01:00,DT#2028-03-26-01:00,DT#2029-03-25-01:00,DT#2030-03-31-01:00];
	aOctober:	ARRAY [2011..2030] OF DT	:=	[DT#2011-10-30-01:00,DT#2012-10-28-01:00,DT#2013-10-27-01:00,DT#2014-10-26-01:00,DT#2015-10-25-01:00,
											DT#2016-10-30-01:00,DT#2017-10-29-01:00,DT#2018-10-28-01:00,DT#2019-10-27-01:00,DT#2020-10-25-01:00,
											DT#2021-10-31-01:00,DT#2022-10-30-01:00,DT#2023-10-29-01:00,DT#2024-10-27-01:00,DT#2025-10-26-01:00,
											DT#2026-10-25-01:00,DT#2027-10-31-01:00,DT#2028-10-29-01:00,DT#2029-10-28-01:00,DT#2030-10-27-01:00];
	tInterval: 		TIME := T#1s; 			(*Częstotliwość aktualizacji czasu*)
END_VAR

t1(IN:= NOT t1.Q, PT:= tInterval);
(* Obliczenia raz na sekunde lub podczas inicjalizacji*)
IF t1.Q THEN
	(* konwersja aktualnego czasy GMT na DWORD *)
	dwActualTime := DT_TO_DWORD(dtActualTimeGMT);
	dwYear := dwActualTime/31536000 + 1970; (* Obliczenie roku *)
	bError := (dwYear<2011) OR (dwYear > 2030); (* jesli jestesmy poza obszarem dzialania blocza - ustawiamy flage bledu *)
	dwActualTime := dwActualTime + 3600; (* czas zimowy GMT + 1 (UTC + 1) *)
	(*czas letni *)
	bSummerTime := (dtActualTimeGMT > aMarch[dwYear]) AND (dtActualTimeGMT < aOctober[dwYear]);
	IF bSummerTime THEN dwActualTime := dwActualTime + 3600; END_IF
	dtActualTimeCET := DWORD_TO_DT(dwActualTime);
END_IF

END_FUNCTION_BLOCK

// ---- POUs/DateAndTime/FB_GetSystemTime.TcPOU
(****************************************************************************************)
(*							Beckhoff Automation Poland									*)
(*								FB_GetSystemTime  v1.2									*)
(*									26.07.2013											*)
(*		v1.2 - zmiana nazwy bloku z FB_Time na FB_GetSystemTime, dodanie wyjscia DT		*)
(*		v1.1 - dodano na wyjściu zmienną czasu w formie struktury TIMESTRUCT 			*)
(*				Blok funkcyjny podający dokładną datę w odrębnych zmiennych				*)
(*						może być wywołany raz w programie PLC							*)
(*						Wymaga dodania biblioteki TcUtilities.lib						*)
(*______________________________________________________________________________________*)
FUNCTION_BLOCK FB_GetSystemTime
VAR_INPUT
	bEnable:			BOOL;				(*Aktywuje pobieranie czasu systemowego*)
END_VAR
VAR_OUTPUT
	stActTime			:	TIMESTRUCT;
	dtActTime: DT;
(*Poszczególne składowe daty*)
	wYear 				:	WORD;
	wMonth 				:	WORD;
	wDayOfWeek 			: 	WORD;
	wDay 				:	WORD;
	wHour 				:	WORD;
	wMinute 			:	WORD;
	wSecond 			:	WORD;
	wMilliseconds 		: 	WORD;
END_VAR
VAR
	fbGetTime			:	NT_GetTime;
	Get					:	TON;
END_VAR
VAR CONSTANT
	tFrequency			:	TIME			:= T#1s;				(*Częstotliwość pobierania czasu*)
END_VAR

Get(IN:= NOT Get.Q AND bEnable, PT:=tFrequency);
fbGetTime(
	NETID:= '',
	START:= Get.Q,
	TMOUT:= T#200ms,
	TIMESTR=>stActTime);

dtActTime 		:= SYSTEMTIME_TO_DT(stActTime);
wDay 			:= stActTime.wDay;
wDayOfWeek 	:= stActTime.wDayOfWeek;
wHour 			:= stActTime.wHour;
wMilliseconds 	:= stActTime.wMilliseconds;
wMinute 		:= stActTime.wMinute;
wMonth 		:= stActTime.wMonth;
wSecond 		:= stActTime.wSecond;
wYear 			:= stActTime.wYear;

END_FUNCTION_BLOCK

// ---- POUs/DateAndTime/FB_Period.TcPOU
(****************************************************************************************)
(*							Beckhoff Automation Poland									*)
(*								FB_Period v1.1											*)
(*									20.02.2008											*)
(*		Blok funkcyjny wystawiający wyjście w określonym przedziale czasu				*)
(*				wymaga podania aktualnego czasu na wejście bloku 						*)
(*																						*)
(*______________________________________________________________________________________*)
FUNCTION_BLOCK FB_Period
VAR_INPUT
	bReset				:	BOOL;									(*Przywrócenie wartości w bloku do stanu początkowego*)
	wStartHour			:	WORD;									(*Godzina wystawienia wyjścia*)
	wStartMinute		:	WORD;									(*Minuta wystawienia wyjścia*)
	wStopHour			:	WORD;									(*Godzina wyzerowania wyjścia*)
	wStopMinute			:	WORD;									(*Minuta  wyzerowania wyjścia*)
	stActTime			:	TIMESTRUCT;								(*Aktualny czas w formie struktury*)
END_VAR
VAR_OUTPUT
	bOut				:	BOOL;									(*Wyjście*)
END_VAR
VAR
	StartEdge			:	R_TRIG;
	StopEdge			:	R_TRIG;
	ResetEdge			:	R_TRIG;
	bFirstCycle			:	BOOL:=TRUE;
	wStartHourOld		: 	WORD;
	wStartMinuteOld		: 	WORD;
	wStopHourOld		: 	WORD;
	wStopMinuteOld		: 	WORD;
END_VAR

StartEdge();
StopEdge();
ResetEdge(CLK:=bReset);

IF ResetEdge.Q THEN
	bOut:=FALSE;
	bFirstCycle:=TRUE;
END_IF;

(*Sprawdzenie czy była zmiana zadanych przedziałów czasowych*)
IF wStartHour<>wStartHourOld OR wStartMinute<>wStartMinuteOld OR wStopHour<>wStopHourOld OR wStopMinute<>wStopMinuteOld THEN
	bFirstCycle:=TRUE;
END_IF;

IF stActTime.wYear <> 0 THEN
	IF bFirstCycle THEN
	(*W pierwszym cylku należy sprawdzić czy włączamy czy wyłączamy i likwidujemy zmienna pierwszego cyklu*)
		IF stActTime.wHour< wStartHour OR stActTime.wHour>wStopHour THEN
		(*Poznajemy po godzinie, ze na pewno jest wylaczone *)
			bOut := FALSE;
		ELSIF (stActTime.wHour=wStartHour AND stActTime.wMinute < wStartMinute) OR (stActTime.wHour=wStopHour AND stActTime.wMinute > wStopMinute)  THEN
		(*W tej godzinie zaczyna sie badz konczy wylaczenie, ale jescze jest wylaczone*)
			bOut := FALSE; (*Wylaczone*)
		ELSE
			bOut := TRUE; (*Wlaczone*)
		END_IF
		bFirstCycle := FALSE;
	ELSE
	(*Teraz reagujemy tylko na zmiany - wykrycie sygnału do startu i końca*)
		StartEdge.CLK := wStartHour = stActTime.wHour AND wStartMinute = stActTime.wMinute;
		StopEdge.CLK := wStopHour = stActTime.wHour AND wStopMinute = stActTime.wMinute;
		IF StartEdge.Q  THEN bOut := TRUE; (*Dzien*) END_IF
		IF StopEdge.Q  THEN bOut := FALSE; (*Noc*) END_IF
	END_IF
END_IF

wStartHourOld:=wStartHour;
wStartMinuteOld:=wStartMinute;
wStopHourOld:=wStopHour;
wStopMinuteOld:=wStopMinute;

END_FUNCTION_BLOCK

// ---- POUs/DateAndTime/FB_PolishPublicHoliday.TcPOU
(************************************************************************************)
(*						Beckhoff Automation Poland								 	*)
(*						FB_PolishPublicHoliday v 1.0								*)
(*							26.07.2013												*)
(*	Blok Funkcyjny ktorego wyjscie jest TRUE w przypadku swieta						*)
(* 			wyjscie stNextHoliday podaje nastepne swieto							*)
(*__________________________________________________________________________________*)
FUNCTION_BLOCK FB_PolishPublicHoliday
VAR_INPUT
	bEnable 			: 			BOOL; 							(*zmienna włączająca bloczek*)
	stActTime 			:			TIMESTRUCT;						(*struktura przechowująca aktualny czas*)
END_VAR
VAR_OUTPUT
	bHoliday 			:	BOOL;									(*zmienna zwracająca TRUE gdy dzisiaj jest swięto*)
	bError				:	BOOL;									(*zmienna błędu*)
	stNextHoliday		:	TIMESTRUCT;								(*zmienna przechowująca datę nastepnego święta*)
END_VAR
VAR
	wNextEasterYear		:	WORD; 									(*Rok najbliższego święta Wielkiej Nocy*)
	bInit				:	BOOL			:=TRUE;					(*zmienna inicjalizująca pierwszy cykl programu*)
	arrHolidays 		:	ARRAY [1..13] OF TIMESTRUCT;   			(*Pomocnicza tablica z swietami Polskimi w danym roku*)
	stEasterDate1		:	TIMESTRUCT;								(*Czas pierwszego dnia świąt w formie struktury*)
	stEasterDate2		:	TIMESTRUCT; 							(*Czas drugiego dnia świąt w formie struktury*)
	stZielSw			:	TIMESTRUCT; 							(*Czas Zielonych Świątek w formie struktury*)
	stBCDate			:	TIMESTRUCT;								(*Czas Bożego Ciała świąt w formie struktury*)
	stTemp				:	TIMESTRUCT;								(*zmienna pomocnicza pomagająca w przesuwaniu tablicy*)
	iCount				:	INT;									(*zmienna pomocnicza inkremetnowana w pętli FOR*)
END_VAR

bError:=stActTime.wYear<2000;
IF bInit AND NOT bError THEN
	wNextEasterYear:=stActTime.wYear;(*ustawienie roku bieżącego jako roku kolejnej Wielkiej Nocy*)
	a_Easter();(*akcja obliczania po kolei świąt ruchomych*)
	a_Easter2();
	a_BC();
	a_ZielSwiatki();
	bInit:=FALSE;(*warunek wejścia do pierwszego cyklu programu nie będzie już spełniony*)
	arrHolidays[1].wDay:=1;(*wyliczenie pierwszy raz na sztywno wszystkich świąt w danym roku  aby znaleźć najbliższe święto*)
	arrHolidays[1].wMonth:=1;
	arrHolidays[1].wYear:=stActTime.wYear;
	arrHolidays[2].wDay:=6;
	arrHolidays[2].wMonth:=1;
	arrHolidays[2].wYear:=stActTime.wYear;
	arrHolidays[3].wDay:=stEasterDate1.wDay;
	arrHolidays[3].wMonth:=stEasterDate1.wMonth;
	arrHolidays[3].wYear:=stEasterDate1.wYear;
	arrHolidays[4].wDay:=stEasterDate2.wDay;
	arrHolidays[4].wMonth:=stEasterDate2.wMonth;
	arrHolidays[4].wYear:=stEasterDate2.wYear;
	arrHolidays[5].wDay:=1;
	arrHolidays[5].wMonth:=5;
	arrHolidays[5].wYear:=stActTime.wYear;
	arrHolidays[6].wDay:=3;
	arrHolidays[6].wMonth:=5;
	arrHolidays[6].wYear:=stActTime.wYear;
	arrHolidays[7].wDay:=stZielSw.wDay;
	arrHolidays[7].wMonth:=stZielSw.wMonth;
	arrHolidays[7].wYear:=stZielSw.wYear;
	arrHolidays[8].wDay:=stBCDate.wDay;
	arrHolidays[8].wMonth:=stBCDate.wMonth;
	arrHolidays[8].wYear:=stBCDate.wYear;
	arrHolidays[9].wDay:=15;
	arrHolidays[9].wMonth:=8;
	arrHolidays[9].wYear:=stActTime.wYear;
	arrHolidays[10].wDay:=1;
	arrHolidays[10].wMonth:=11;
	arrHolidays[10].wYear:=stActTime.wYear;
	arrHolidays[11].wDay:=11;
	arrHolidays[11].wMonth:=11;
	arrHolidays[11].wYear:=stActTime.wYear;
	arrHolidays[12].wDay:=25;
	arrHolidays[12].wMonth:=12;
	arrHolidays[12].wYear:=stActTime.wYear;
	arrHolidays[13].wDay:=26;
	arrHolidays[13].wMonth:=12;
	arrHolidays[13].wYear:=stActTime.wYear;

	stNextHoliday := arrHolidays[1];		(*przypisanie wartości stNextHoliday na 1. stycznia bieżącego roku*)

	(*i porównywanie tej daty do daty obecnej*)
	WHILE stActTime.wYear = stNextHoliday.wYear AND (stActTime.wMonth>stNextHoliday.wMonth OR (stActTime.wDay>stNextHoliday.wDay)) DO
		a_MoveArray();		(*w celu przesunięcia tablicy tak, aby pierwszy element był najbliższym świętem*)
	END_WHILE
END_IF

(*instrukcja warunkowa przesuwająca tablicę, o ile data stNextHoliday minęła*)
IF stActTime.wYear > stNextHoliday.wYear OR (stActTime.wYear = stNextHoliday.wYear AND (stActTime.wMonth>stNextHoliday.wMonth OR (stActTime.wMonth = stNextHoliday.wMonth AND stActTime.wDay>stNextHoliday.wDay))) THEN
	a_MoveArray();
END_IF

(*przypisanie wartości wyjścia typu bool; wartość równa 1 gdy obecna data jest datą najbliższego święta*)
bHoliday := (stActTime.wYear = stNextHoliday.wYear) AND (stActTime.wMonth = stNextHoliday.wMonth) AND (stActTime.wDay = stNextHoliday.wDay);

ACTION a_BC:
(*Wyliczenie daty Bożego Ciała /z przypisaniem do stBCDate/*)
stBCDate.wMonth := stEasterDate1.wMonth+2;
stBCDate.wDay := stEasterDate1.wDay -1;
IF stBCDate.wDay = 0 THEN
	stBCDate.wMonth := 5;
	stBCDate.wDay := 31;
END_IF
stBCDate.wYear := stEasterDate1.wYear;
END_ACTION

ACTION a_Easter:
(*Akcja służąca do wyliczania daty Wielkiejnocy /z przypisaniem do stEasterDate1/*)
stEasterDate1.wDay :=  ((((19*(wNextEasterYear MOD 19)+(wNextEasterYear/100)-((wNextEasterYear/100)/4)-(((wNextEasterYear/100)-(((wNextEasterYear/100)+8)/25)+1)/3)+15) MOD 30)+((32+2*((wNextEasterYear/100) MOD 4)+2*((wNextEasterYear MOD 100)/4)-((19*(wNextEasterYear MOD 19)+(wNextEasterYear/100)-((wNextEasterYear/100)/4)-(((wNextEasterYear/100)-(((wNextEasterYear/100)+8)/25)+1)/3)+15) MOD 30)-((wNextEasterYear MOD 100) MOD 4)) MOD 7)-7*(((wNextEasterYear MOD 19)+11*((19*(wNextEasterYear MOD 19)+(wNextEasterYear/100)-((wNextEasterYear/100)/4)-(((wNextEasterYear/100)-(((wNextEasterYear/100)+8)/25)+1)/3)+15) MOD 30)+22*((32+2*((wNextEasterYear/100) MOD 4)+2*((wNextEasterYear MOD 100)/4)-((19*(wNextEasterYear MOD 19)+(wNextEasterYear/100)-((wNextEasterYear/100)/4)-(((wNextEasterYear/100)-(((wNextEasterYear/100)+8)/25)+1)/3)+15) MOD 30)-((wNextEasterYear MOD 100) MOD 4)) MOD 7))/451)+114) MOD 31)+1;
stEasterDate1.wMonth:=  (((19*(wNextEasterYear MOD 19)+(wNextEasterYear/100)-((wNextEasterYear/100)/4)-(((wNextEasterYear/100)-(((wNextEasterYear/100)+8)/25)+1)/3)+15) MOD 30)+((32+2*((wNextEasterYear/100) MOD 4)+2*((wNextEasterYear MOD 100)/4)-((19*(wNextEasterYear MOD 19)+(wNextEasterYear/100)-((wNextEasterYear/100)/4)-(((wNextEasterYear/100)-(((wNextEasterYear/100)+8)/25)+1)/3)+15) MOD 30)-((wNextEasterYear MOD 100) MOD 4)) MOD 7)-7*(((wNextEasterYear MOD 19)+11*((19*(wNextEasterYear MOD 19)+(wNextEasterYear/100)-((wNextEasterYear/100)/4)-(((wNextEasterYear/100)-(((wNextEasterYear/100)+8)/25)+1)/3)+15) MOD 30)+22*((32+2*((wNextEasterYear/100) MOD 4)+2*((wNextEasterYear MOD 100)/4)-((19*(wNextEasterYear MOD 19)+(wNextEasterYear/100)-((wNextEasterYear/100)/4)-(((wNextEasterYear/100)-(((wNextEasterYear/100)+8)/25)+1)/3)+15) MOD 30)-((wNextEasterYear MOD 100) MOD 4)) MOD 7))/451)+114)/31;
stEasterDate1.wYear := wNextEasterYear;

wNextEasterYear := stEasterDate1.wYear+1;
END_ACTION

ACTION a_Easter2:
(*Obliczenie drugiego dnia Wielkiejnocy /przypisanie do stEasterDate2/*)
IF stEasterDate1.wDay=31 THEN
	stEasterDate2.wDay:=1;
	stEasterDate2.wMonth:=4;
ELSE
	stEasterDate2.wDay:=stEasterDate1.wDay+1;
	stEasterDate2.wMonth:=stEasterDate1.wMonth;
END_IF
stEasterDate2.wYear := stEasterDate1.wYear;
END_ACTION

ACTION a_MoveArray:
(*Akcja przesuwająca tablicę świąt. Dodatkowo za pomocą tej akcji obliczana jest data święta z arrHolidays[1] w roku kolejnym*)

IF arrHolidays[1].wYear = stEasterDate1.wYear AND arrHolidays[1].wMonth = stEasterDate1.wMonth AND arrHolidays[1].wDay = stEasterDate1.wDay THEN
	a_Easter();						(*Dla świąt ruchomych obliczana jest nowa data; Wielkanoc*)
	arrHolidays[1] := stEasterDate1;
ELSIF arrHolidays[1].wYear = stEasterDate2.wYear AND arrHolidays[1].wMonth = stEasterDate2.wMonth AND arrHolidays[1].wDay = stEasterDate2.wDay THEN
	a_Easter2();						(*Drugi dzień świąt*)
	arrHolidays[1] := stEasterDate2;
ELSIF arrHolidays[1].wYear = stZielSw.wYear AND arrHolidays[1].wMonth = stZielSw.wMonth AND arrHolidays[1].wDay = stZielSw.wDay THEN
	a_ZielSwiatki();						(*Zielone świątki*)
	arrHolidays[1] := stZielSw;
ELSIF arrHolidays[1].wYear = stBCDate.wYear AND arrHolidays[1].wMonth = stBCDate.wMonth AND arrHolidays[1].wDay = stBCDate.wDay THEN
	a_BC();							(*Boż Ciało*)
	arrHolidays[1] := stBCDate;
ELSE								(*Jeżeli jest to święto stałe, dodawany jest tylko rok*)
	arrHolidays[1].wYear := arrHolidays[1].wYear+1;
END_IF;

(*Następnie elementy tablicy są przesuwane; Pierwszy element tablicy (po zapisaniu do stTemp) idzie na koniec tablicy (arrHolidays[13]); Reszta elementów przesuwa się o 1 wyżej*)
stTemp := arrHolidays[1];
FOR iCount := 1 TO 12 DO
	arrHolidays[iCount] := arrHolidays[iCount+1];
END_FOR
arrHolidays[13] := stTemp;

(*wpisanie poprawnej wartości najbliższego święta do stNextHoliday*)
stNextHoliday := arrHolidays[1];
END_ACTION

ACTION a_ZielSwiatki:
(*Akcja służąca do obliczania daty Zielonych Świątek /w strukturze stZielSw/*)
IF stEasterDate1.wMonth =3 THEN
	stZielSw.wMonth := 5;
	stZielSw.wDay := stEasterDate1.wDay-12;
ELSIF stEasterDate1.wDay < 13 THEN
	stZielSw.wMonth := 5;
	stZielSw.wDay := stEasterDate1.wDay+19;
ELSE
	stZielSw.wMonth := 6;
	stZielSw.wDay := stEasterDate1.wDay-12;
END_IF
stZielSw.wYear := stEasterDate1.wYear;
END_ACTION

END_FUNCTION_BLOCK

// ---- POUs/DateAndTime/FB_SimpleWorkTime.TcPOU
//==================================================================================================
//							Beckhoff Automation Poland
//									30.03.2017
//	Proste zliczanie czasu pracy, podaje czas aktualnego zalaczenia, ostatniego zalaczenia, sumarycznego zalaczenia
// 	v1.0	|| TC v 3.1.4020.32		|| - pierwsza wersja
//==================================================================================================
FUNCTION_BLOCK FB_SimpleWorkTime
VAR_INPUT
	bIn										: BOOL;
	bReset									: BOOL;					// Zerowanie wartosci
END_VAR
VAR_OUTPUT
	tCurrentTime							: TIME;					// Aktualny czas zalaczenia
	tLastTime								: TIME;					// Ostatni czas zalaczenia
	tSummaryTime							: TIME;					// Sumaryczny czas zalaczenia
END_VAR
VAR
	fbTimeMeasure							: FB_TimeMeasureEx;		// Licznik czasu
	tLastSummaryTime						: TIME;					// Zmienna do wewnetrznych przeliczen
END_VAR

fbTimeMeasure(bOn:= bIn, bReset := bReset, tCurrentTime=> tCurrentTime, tLastTime=> tLastTime);
IF bIn THEN
	tSummaryTime 		:= tLastSummaryTime + tCurrentTime;
ELSE
	tLastSummaryTime 	:= tSummaryTime;
END_IF

IF bReset THEN
	tSummaryTime 		:= T#0S;
	tLastSummaryTime 	:= T#0S;
END_IF

END_FUNCTION_BLOCK

// ---- POUs/DateAndTime/FB_TimeMeasureEx.TcPOU
//==================================================================================================
//							Beckhoff Automation Poland
//									30.03.2017
//		Mierzy czas zalaczenia wejscia. Podaje aktualny czas oraz czas ostatniego zalaczenia
//		W porownaniu do FB_TimeMeasure ma wejscie bReset
// 	v1.0 	|| TC v 3.1.4020.32		|| - pierwsza wersja
//==================================================================================================
FUNCTION_BLOCK FB_TimeMeasureEx
VAR_INPUT
	bOn										: BOOL;					// Zliczany sygnal
	bReset									: BOOL;					// Zerowanie wartosci
END_VAR
VAR_OUTPUT
	tCurrentTime							: TIME;
	tLastTime								: TIME;
END_VAR
VAR
	ton1									: TON;
	bOnOld									: BOOL;
END_VAR

IF bOn = FALSE AND bOnOld = TRUE THEN 
	tLastTime := tCurrentTime; 
END_IF
ton1(IN:= bOn, PT:= T#71582m47s295ms, Q=> , ET=> tCurrentTime);
bOnOld 						:= bOn;
IF bReset THEN
	bOnOld					:= FALSE;
	tLastTime				:= T#0S;
	tCurrentTime			:= T#0S;
	ton1(IN:= FALSE);
END_IF

END_FUNCTION_BLOCK

// ---- POUs/DateAndTime/FB_TimeMeasure.TcPOU
(****************************************************************************************)
(*							Beckhoff Automation Poland									*)
(*								FB_TimeMeasure v1.1										*)
(*									13.08.2012											*)
(* Mierzy czas załączenia wejścia. Podaje aktualny czas oraz czas ostatniego załączenia *)
(*______________________________________________________________________________________*)
FUNCTION_BLOCK FB_TimeMeasure
VAR_INPUT
	bOn				:	BOOL;
END_VAR
VAR_OUTPUT
	tCurrentTime	:	TIME;
	tLastTime		:	TIME;
END_VAR
VAR
	ton1			:	TON;
	bOnOld			:	BOOL;
END_VAR

IF bOn = FALSE AND bOnOld = TRUE THEN tLastTime := tCurrentTime; END_IF
ton1(IN:= bOn, PT:= T#71582m47s295ms, Q=> , ET=> tCurrentTime);
bOnOld := bOn;

END_FUNCTION_BLOCK

// ---- POUs/DateAndTime/FB_WeekSchedule.TcPOU
(****************************************************************************************)
(*							Beckhoff Automation Poland									*)
(*								FB_WeekSchedule  v1.2									*)
(*									24.05.2011											*)
(*		Blok funkcyjny wystawiający wyjście w określonych przedziałach czasu			*)
(*				wymaga podania aktualnego czasu na wejście bloku 						*)
(*																						*)
(*______________________________________________________________________________________*)
FUNCTION_BLOCK FB_WeekSchedule
VAR_INPUT
	bReset:				BOOL;				(*Przywrócenie wartości w bloku do stanu początkowego*)
	wStartHour:			WORD;				(*Godzina wystawienia wyjścia*)
	wStartMinute:		WORD;				(*Minuta wystawienia wyjścia*)
	wStopHour:			WORD;				(*Godzina wyzerowania wyjścia*)
	wStopMinute:		WORD;				(*Minuta  wyzerowania wyjścia*)
	
	(*Dni tygodnia w których ma działać blok funkcyjny*)
	bMonday: 			BOOL;
	bTuesday:			BOOL;
	bWednesday:			BOOL;
	bThursday:			BOOL;
	bFriday:			BOOL;
	bSaturday:			BOOL;
	bSunday:			BOOL;
	stActTime: 			TIMESTRUCT;			(*Aktualny czas w formie struktury*)
END_VAR
VAR_OUTPUT
	bOut:				BOOL;				(*Wyjście*)
	bEdgeOn:	 		BOOL;				(* wystawia true na jeden cykl gdy zadanie rozpoczyna się wykonywać *)
	bEdgeOff: 			BOOL;				(* wystawia true na jeden cykl gdy zadanie konczy się wykonywac *)
END_VAR
VAR
	StartEdge:			R_TRIG;
	StopEdge:			R_TRIG;
	ResetEdge:			R_TRIG;
	EdgeOn:				R_TRIG;
	EdgeOff:			F_TRIG;
	bGo: 				BOOL;
	bFirstCycle:		BOOL	:=TRUE;
	wStartHourOld: 		WORD;
	wStartMinuteOld: 	WORD;
	wStopHourOld: 		WORD;
	wStopMinuteOld: 	WORD;
END_VAR

StartEdge();
StopEdge();
ResetEdge(CLK:=bReset);
IF ResetEdge.Q THEN
	bOut:=FALSE;
	bFirstCycle:=TRUE;
END_IF;

CASE stActTime.wDayOfWeek OF
	0:	bGo := bSunday;
	1:	bGo := bMonday;
	2:	bGo := bTuesday;
	3:	bGo := bWednesday;
	4:	bGo := bThursday;
	5:	bGo := bFriday;
	6:	bGo := bSaturday;
END_CASE

(*Sprawdzenie czy była zmiana zadanych przedziałów czasowych*)
IF wStartHour<>wStartHourOld OR wStartMinute<>wStartMinuteOld OR wStopHour<>wStopHourOld OR wStopMinute<>wStopMinuteOld THEN
	bFirstCycle:=TRUE;
END_IF;

IF bGo AND stActTime.wYear <> 0 THEN
	IF bFirstCycle THEN
	(*W pierwszym cylku należy sprawdzić czy włączamy czy wyłączamy i likwidujemy zmienna pierwszego cyklu*)
		IF stActTime.wHour< wStartHour OR stActTime.wHour>wStopHour THEN
		(*Poznajemy po godzinie, ze na pewno jest wylaczone *)
			bOut := FALSE;
		ELSIF (stActTime.wHour=wStartHour AND stActTime.wMinute < wStartMinute) OR (stActTime.wHour=wStopHour AND stActTime.wMinute > wStopMinute)  THEN
		(*W tej godzinie zaczyna sie badz konczy wylaczenie, ale jescze jest wylaczone*)
			bOut := FALSE; (*Wylaczone*)
		ELSE
			bOut := TRUE; (*Wlaczone*)
		END_IF
		bFirstCycle := FALSE;
	ELSE
		(*Sprawdzamy czy zdarzenie jest całodniowe*)
		IF wStartHour=0 AND wStartMinute=0 AND wStopHour=0 AND wStopMinute=0 THEN
			bOut := TRUE; (*Dzien*)
		END_IF
		(*Teraz reagujemy tylko na zmiany - wykrycie sygnału do startu i końca*)
		StartEdge.CLK := wStartHour = stActTime.wHour AND wStartMinute = stActTime.wMinute;
		StopEdge.CLK := wStopHour = stActTime.wHour AND wStopMinute = stActTime.wMinute;
		IF StartEdge.Q  THEN bOut := TRUE; (*Dzien*) END_IF
		IF StopEdge.Q  THEN bOut := FALSE; (*Noc*) END_IF
	END_IF
ELSE
	bOut := FALSE;
	StartEdge.CLK := FALSE;
	StopEdge.CLK := FALSE;
END_IF
(*Wartości wystawione na 1 cykl*)
EdgeOn(CLK:= bOut, Q=>bEdgeOn );
EdgeOff(CLK:= bOut, Q=>bEdgeOff );

wStartHourOld:=wStartHour;
wStartMinuteOld:=wStartMinute;
wStopHourOld:=wStopHour;
wStopMinuteOld:=wStopMinute;

END_FUNCTION_BLOCK

// ---- POUs/DateAndTime/FB_Worktime.TcPOU
(********************************************************************************************************)
(*							Beckhoff Automation Poland													*)
(*								FB_Worktime  v3															*)
(*									3.11.2011															*)
(*							v3 - unifikacja wejść i wyjść, przejście z j. polskiego na j. angielski		*)
(*	Bloczek zliczajacy czas zalaczenia wejscia bInput													*)
(*	Pozwala zadac wartosc startowa czasu lub dodac dowolna wartosc do mierzonego czasu					*)
(*	Zliczony czas podaje w postaci sumarycznej liczy minut lub z podzialem na poszczegolne skladowe		*)
(*	Posiada możliwość wpisania czasu (limitu), którego upłynięcie będzie sygnalizowane wyjściem  bLimit	*)
(*______________________________________________________________________________________________________*)
FUNCTION_BLOCK FB_Worktime
VAR_INPUT
	bInput : 			BOOL;				(*Gdy bInput = TRUE to zliczamy czas*)
	bAdd : 				BOOL;				(*Dodanie do sumarycznego czasu wartości z wStartwDzien, wStartwGodz i wStartMinute*)
	bReset :	 		BOOL;				(*Ustawienie jako czas sumaryczny wartosci wStartwDzien, wStartwGodz i wStartMinute*)
	wStartDay: 			WORD;				(*Dodawana/ustawiana podczas resetu liczba dni*)
	wStartHour: 		WORD;				(*Dodawana/ustawiana podczas resetu  liczba godzin*)
	wStartMinute: 		WORD;				(*Dodawana/ustawiana podczas resetu liczba minut*)
	wDaysLimit:			WORD;				(*Wprowadzanie limitu dni*)
	wHoursLimit:		WORD;				(*Wprowadzanie limitu godzin*)
	wMinutesLimit:		WORD;				(*Wprowadzanie limitu min*)
END_VAR
VAR_OUTPUT
	bLimit:				BOOL;				(* Pokazuje czy upłynął zadany czas*)
END_VAR
VAR_IN_OUT
	dwSummaryMinutes: 	DWORD;				(*Czas sumaryczny w minutach*)
	wDays:				WORD;				(*Podzial na czesci*)
	wHours:				WORD;
	wMinutes:			WORD;
END_VAR
VAR
	Odliczanie_Czasu: 	TON; 				(*Glowny timer liczacy*)
	Obliczenia: 		TON; 				(*Timer ustalajacy co ile wykonywane sa obliczenia*)
	rtDodaj: 			R_TRIG; 			(*Wyzwalanie dodania wartosci*)
	rtReset: 			R_TRIG; 			(*Wyzwalanie resetu licznika*)
	ftKoniecPracy: 		F_TRIG; 			(*Wykrycie konca zliczanego sygnalu*)
	tET: 				TIME; 				(*Czas ktory uplynal od ostatniego zalaczenia sygnalu*)
	bFirstCycle: 		BOOL	:=TRUE;		(*Flaga pierwszego cyklu*)
	(*Aktualnie dodawany czas*)
	wDodatkoweMinuty : 	WORD;
	wDodatkoweGodziny : WORD;
	wDodatkoweDni : 	WORD;
	wMiliSek: 			DWORD;
	(*Ostatnio zapisane wartosci*)
	wMinOld: 			WORD;
	wGodzOld: 			WORD;
	wDzienOld: 			WORD;
	dwSumMinOld: 		DWORD;
	wMiliSekOld: 		DWORD;
	(*Limit*)
	wMinLimit:			WORD;
	wGodzLimit:			WORD;
	wDzienLimit:		WORD;
	wMinOldLimit:		WORD;
	wGodzOldLimit:		WORD;
	wDzienOldLimit:		WORD;
	wLimitDzienOld:		WORD;
	wLimitGodzOld:		WORD;
	wLimitMinOld:		WORD;

END_VAR

(*Wpisanie wartosci z podtrzymania zasialnia*)
	IF bFirstCycle THEN
		wDzienOld := wDays;
		wGodzOld := wHours;
		wMinOld := wMinutes;
		dwSumMinOld := dwSummaryMinutes;
		bFirstCycle := FALSE;
	END_IF
(*Dodanie wartosci startowej*)
	rtDodaj(CLK:=bAdd );
	IF rtDodaj.Q THEN
		wDodatkoweGodziny := ((wMinOld + wStartMinute) -((wMinOld + wStartMinute) MOD 60))/60;(*Obliczenie dodatkowych godzin*)
		wDodatkoweDni := ((wGodzOld + wStartHour + wDodatkoweGodziny) -((wGodzOld + wStartHour + wDodatkoweGodziny )MOD 24))/24;(*Obliczenie dodatkowych dni*)
		wDzienOld := wDzienOld + wStartDay + wDodatkoweDni;(*Obliczenie dni*)
		wGodzOld := (wGodzOld + wStartHour + wDodatkoweGodziny) MOD 24; (*Dodanie godzin, jeżeli więcej niż 24, to dodanie zostanie to do dni*)
		wMinOld := (wMinOld + wStartMinute) MOD 60; (*Dodanie minut, jeżeli więcej niż 60, to dodanie zostanie to do godziny*)
		dwSumMinOld := dwSumMinOld + wStartDay*1440 + wStartHour*60 + wStartMinute; (*24*60 = 1440*)
		wDays := wDzienOld; (*Przepisanie obliczen na wyjscia*)
		wHours := wGodzOld;
		wMinutes := wMinOld;
		dwSummaryMinutes:= dwSumMinOld;
	END_IF
(*Reset licznika*)
	rtReset(CLK:= bReset);
	IF rtReset.Q THEN
		wDodatkoweGodziny := (wStartMinute -(wStartMinute MOD 60))/60;(*Obliczenie dodatkowych godzin*)
		wDodatkoweDni := ((wStartHour + wDodatkoweGodziny) -((wStartHour + wDodatkoweGodziny) MOD 24))/24;(*Obliczenie dodatkowych godzin*)
		wDzienOld := wStartDay + wDodatkoweDni;(*Dodanie sumarycznego*)
		wGodzOld := (wStartHour + wDodatkoweGodziny) MOD 24; (*Dodanie godzin, jeżeli więcej niż 24, to dodanie zostanie to do dni*)
		wMinOld := wStartMinute MOD 60; (*Dodanie minut, jeżeli więcej niż 60, to dodanie zostanie to do godziny*)
		dwSumMinOld := wStartDay*1440 + wStartHour*60 + wStartMinute;(*24*60 = 1440*)
		wDays := wDzienOld;(*Przepisanie obliczen na wyjscia*)
		wHours := wGodzOld;
		wMinutes := wMinOld;
		dwSummaryMinutes:= dwSumMinOld;
	END_IF

(*Zliczanie czasu pracy*)
	ftKoniecPracy(CLK:= bInput OR Odliczanie_Czasu.Q, Q=> );
	Odliczanie_Czasu(IN:= (bInput AND NOT Odliczanie_Czasu.Q AND NOT bReset) OR ftKoniecPracy.Q, PT:= T#24h, ET=> tET);
	Obliczenia(IN:= NOT Obliczenia.Q, PT:= T#59s); (*Aby nie liczyc caly czas*)
	IF ftKoniecPracy.Q THEN
		wMiliSek := TIME_TO_DWORD(tET) + wMiliSekOld;
		wDodatkoweMinuty := DWORD_TO_WORD(wMiliSek/60000) MOD 60; (*Obliczenie dodatkowych minut*)
		wDodatkoweGodziny := DWORD_TO_WORD(wMiliSek/3600000) MOD 24; (*Obliczenie dodatkowych godzin 60 000*60 = 3 600 000*)
		wDodatkoweDni := DWORD_TO_WORD(wMiliSek/86400000);(*Obliczenie dodatkowych dni 60000*60*24 = 86 400 000*)

		wMinutes := (wMinOld + wDodatkoweMinuty) MOD 60;
		wHours := (wGodzOld + wDodatkoweGodziny + ((wMinOld + wDodatkoweMinuty) - wMinutes)/60) MOD 24; (*Dodanie godzin, jeżeli więcej niż 24, to dodanie zostanie to do dni*)
		wDays := wDzienOld + wDodatkoweDni + ((wGodzOld + wDodatkoweGodziny + ((wMinOld + wDodatkoweMinuty) - wMinutes)/60) - wHours)/24;(*Dodanie sumarycznego*)
		dwSummaryMinutes := dwSumMinOld + DWORD_TO_WORD(wMiliSek/60000);
		(*Przepisanie obliczen na wyjscia*)
		wDzienOld := wDays;
		wGodzOld := wHours;
		wMinOld := wMinutes;
		dwSumMinOld := dwSummaryMinutes;
		wMiliSekOld := wMiliSek MOD 60000; (*Obliczenie ile mili sec zostalo nieuwzglednionych*)
	ELSIF Obliczenia.Q THEN
		wMiliSek := TIME_TO_DWORD(tET) + wMiliSekOld;
		wDodatkoweMinuty := DWORD_TO_WORD(wMiliSek/60000) MOD 60; (*Obliczenie dodatkowych minut*)
		wDodatkoweGodziny := DWORD_TO_WORD(wMiliSek/3600000) MOD 24; (*Obliczenie dodatkowych godzin*)
		wDodatkoweDni := DWORD_TO_WORD(wMiliSek/86400000);(*Obliczenie dodatkowych dni*)
		(*Przepisanie obliczen na wyjscia*)
		wMinutes := (wMinOld + wDodatkoweMinuty) MOD 60;
		wHours := (wGodzOld + wDodatkoweGodziny + ((wMinOld + wDodatkoweMinuty) - wMinutes)/60) MOD 24; (*Dodanie godzin, jeżeli więcej niż 24, to dodanie zostanie to do dni*)
		wDays := wDzienOld + wDodatkoweDni + ((wGodzOld + wDodatkoweGodziny + ((wMinOld + wDodatkoweMinuty) - wMinutes)/60) - wHours)/24;(*Dodanie sumarycznego*)
		dwSummaryMinutes := dwSumMinOld + DWORD_TO_WORD(wMiliSek/60000);
	END_IF

	IF Odliczanie_Czasu.Q THEN wDzienOld := wDzienOld + 1; END_IF (*Reset zegara po dobie, dodajemy 1 dzien*)

(*Dodawanie limitu*)

	IF 	wLimitDzienOld<>wDaysLimit OR wLimitGodzOld<>wHoursLimit OR wLimitMinOld<>wMinutesLimit THEN
		wDodatkoweGodziny := (wMinutesLimit -(wMinutesLimit MOD 60))/60;(*Obliczenie dodatkowych godzin*)
		wDodatkoweDni := ((wHoursLimit + wDodatkoweGodziny) -((wHoursLimit + wDodatkoweGodziny) MOD 24))/24;(*Obliczenie dodatkowych godzin*)
		wDzienOldLimit := wDaysLimit + wDodatkoweDni;(*Dodanie sumarycznego*)
		wGodzOldLimit := (wHoursLimit + wDodatkoweGodziny) MOD 24; (*Dodanie godzin, jeżeli więcej niż 24, to dodanie zostanie to do dni*)
		wMinOldLimit := wMinutesLimit MOD 60; (*Dodanie minut, jeżeli więcej niż 60, to dodanie zostanie to do godziny*)
		wDzienLimit := wDzienOldLimit;(*Przepisanie obliczen na wyjscia*)
		wGodzLimit := wGodzOldLimit;
		wMinLimit := wMinOldLimit;
	END_IF
(*sprawdzanie limitu*)
	IF wDzienLimit<>0 OR wGodzLimit <>0 OR wMinLimit <>0 THEN
		IF wDays > wDzienLimit THEN
			bLimit:=TRUE;
		ELSIF wDays=wDzienLimit THEN
			IF wHours > wGodzLimit THEN
				bLimit:=TRUE;
			ELSIF wHours = wGodzLimit THEN
				IF wMinutes >= wMinLimit THEN
					bLimit:=TRUE;
				ELSE
					bLimit:=FALSE;
				END_IF
			ELSE
				bLimit:=FALSE;
			END_IF
		ELSE
			bLimit:=FALSE;
		END_IF
	END_IF
	wLimitDzienOld:=wDaysLimit;
	wLimitGodzOld:=wHoursLimit;
	wLimitMinOld:=wMinutesLimit;

END_FUNCTION_BLOCK

// ---- POUs/DateAndTime/FB_WorktimeCompact.TcPOU
(****************************************************************************************)
(*							Beckhoff Automation Poland									*)
(*								FB_WorktimeCompact v1.0									*)
(*									31.09.2011											*)
(*							Licznik czasu pracy i liczby załaczeń.						*)
(*			Zmienne IN_OUT powinny być przechowywane po zaniku zasilania				*)
(*______________________________________________________________________________________*)
FUNCTION_BLOCK FB_WorktimeCompact
VAR_INPUT
	bIn			:	BOOL;
END_VAR
VAR_IN_OUT
	dwMinutes	: 	DWORD;
	dwCounts	:	DWORD;
END_VAR
VAR
	Timer		:	TON;
	rtMinute	:	R_TRIG;
	i			:	DWORD;
	iOld		:	DWORD;
	rtOn		:	R_TRIG;
END_VAR

(* Wyciągamy sekundy *)
i := TIME_TO_DWORD(Timer.ET) MOD 60000;

IF bIn THEN
	(* Jak działa to sprawdzamy czy się minuta nie przepętliła *)
	rtMinute(CLK:= iOld>i, Q=> );
ELSE
	(* Jak nie działa to sprawdzamy czy było więcej niż 30 s, jak tak to dodamy minutę *)
	rtMinute(CLK:= i>30000, Q=> );
END_IF
(* Timer odliczający czas *)
Timer(IN:=bIn AND NOT Timer.Q ,PT:= T#24h);
(* Przepisanie poprzednich sekund - do wykrycia przepętlenia *)
iOld := i;
(* Dodanie minuty *)
IF rtMinute.Q THEN
	dwMinutes := dwMinutes+1;
END_IF
(* Licznik załaczeń *)
rtOn(CLK:=bIn);
IF rtOn.Q THEN dwCounts := dwCounts+1; END_IF

END_FUNCTION_BLOCK

// ---- POUs/Various/TIMER.TcPOU
FUNCTION_BLOCK TIMER
VAR_INPUT
	IN 			: BOOL;		// Start input
	RIN			: BOOL;		// Reset input
END_VAR
VAR_OUTPUT
	ET			: TIME;		// Accumulated time
END_VAR
VAR
	startTime 	: TIME;
	inputTrig	: R_TRIG;
	resetTrig	: R_TRIG;
END_VAR

(* Update start time *)
inputTrig(CLK := IN AND NOT RIN);
startTime := SEL(inputTrig.Q, startTime, TIME() - ET); 

(* Reset timer *)
resetTrig(CLK := RIN);
ET := SEL(resetTrig.Q, ET, T#0S);

(* Set output time *)
ET 	:= SEL(IN AND NOT RIN, ET, TIME() - startTime);

END_FUNCTION_BLOCK

// ---- POUs/DateAndTime/F_DT_To_sDT_Ind.TcPOU
(********************************************************************************)
(*							Beckhoff Automation Poland							*)
(*								F_DT_To_sDT_Ind v1.0							*)
(*									15.02.2010									*)
(*		Funkcja konwersji zmiennej DT z TC do formatu daty w Indusoft			*)
(*______________________________________________________________________________*)
FUNCTION F_DT_To_sDT_Ind : STRING
VAR_INPUT
	dtTC	:	DT; (*DT z TC*)
END_VAR
VAR
	sDT_TC	:	STRING(22);
END_VAR

sDT_TC := DT_TO_STRING(dtTC);										(*DT#YYYY-MM-DD-GG:MM:SS*)
F_DT_To_sDT_Ind := MID(sDT_TC,8,15);								(*GG:MM:SS*)
F_DT_To_sDT_Ind := CONCAT('// ', F_DT_To_sDT_Ind);					(*// GG:MM:SS*)
F_DT_To_sDT_Ind := INSERT(F_DT_To_sDT_Ind, MID(sDT_TC,4,4),2);	(*//YYYY GG:MM:SS*)
F_DT_To_sDT_Ind := INSERT(F_DT_To_sDT_Ind, MID(sDT_TC,2,12),1);	(*/DD/YYYY GG:MM:SS*)
F_DT_To_sDT_Ind := CONCAT( MID(sDT_TC,2,9),F_DT_To_sDT_Ind);	(*MM/DD/YYYY GG:MM:SS*)

END_FUNCTION

// ---- POUs/DateAndTime/F_ExcelDateMin.TcPOU
(****************************************************************************************)
(*							Beckhoff Automation Poland									*)
(*								F_ExcelDateMin v1.1										*)
(*									9.11.2007											*)
(*		Funkcja konwerująca strukturę TIMESTRUCT  na zmienną typu STRING(17).			*)
(*		Nowa zmienna zawiera datę dzienną z dokładnością minuty.						*)
(*		Format daty pozwala na bezpośrednie wykorzystanie jej w programie Excel.		*)
(*______________________________________________________________________________________*)

FUNCTION F_ExcelDateMin : STRING(16)
VAR_INPUT
	strCzas		:	TIMESTRUCT;		(*Czas w formie struktury*)
END_VAR

F_ExcelDateMin := SYSTEMTIME_TO_STRING(strCzas);
F_ExcelDateMin := REPLACE (F_ExcelDateMin,' ' ,1,11);(*zamiana znaku "-" na " " przed godziną*)

END_FUNCTION

// ---- POUs/DateAndTime/F_ExcelDateSec.TcPOU
(****************************************************************************************)
(*							Beckhoff Automation Poland									*)
(*								F_ExcelDateSec v1.1										*)
(*									9.11.2007											*)
(*		Funkcja konwerująca strukturę TIMESTRUCT  na zmienną typu STRING(20).			*)
(*		Nowa zmienna zawiera datę dzienną z dokładnością sekundy.						*)
(*		Format daty pozwala na bezpośrednie wykorzystanie jej w programie Excel.		*)
(*______________________________________________________________________________________*)

FUNCTION F_ExcelDateSec : STRING(19)
VAR_INPUT
	strCzas									:	TIMESTRUCT;			(*Czas w formie struktury*)
END_VAR

F_ExcelDateSec  := SYSTEMTIME_TO_STRING(strCzas);
F_ExcelDateSec  := REPLACE (F_ExcelDateSec,' ' ,1,11);(*zamiana znaku "-" na " " przed godziną*)

END_FUNCTION

// ---- POUs/DateAndTime/F_sDT_Ind_To_DT.TcPOU
(****************************************************************************************)
(*							Beckhoff Automation Poland									*)
(*								F_sDT_Ind_To_DT v1.0									*)
(*									15.02.2010											*)
(*					Funkcja konwersji zmiennej DT z Indusoft do TC 						*)
(*______________________________________________________________________________________*)
FUNCTION F_sDT_Ind_To_DT : DT
VAR_INPUT
	sDT_Indusoft			:	STRING;
END_VAR
VAR
	sDT_TC					:	STRING(22);
END_VAR

sDT_TC := CONCAT('DT#',MID(sDT_Indusoft,4,7));		(*DT#YYYY*)
sDT_TC := CONCAT(sDT_TC,'---');						(*DT#YYYY---*)
sDT_TC := INSERT(sDT_TC,MID(sDT_Indusoft,2,1),8);	(*DT#YYYY-MM--*)
sDT_TC := INSERT(sDT_TC,MID(sDT_Indusoft,2,4),11);	(*DT#YYYY-MM-DD-*)
sDT_TC := INSERT(sDT_TC,MID(sDT_Indusoft,8,12),14);	(*DT#YYYY-MM-DD-GG:MM:SS*)
F_sDT_Ind_To_DT := STRING_TO_DT(sDT_TC);

END_FUNCTION

